LIN {X 0,Y 319.792,Z 522.033,A -85,B 0,C 180,E1 -15954.335,E2 -15954.335} C_VEL
LIN {X 0,Y 322.033,Z 507.948,A -85,B 0,C 180,E1 -15955.273,E2 -15955.273} C_VEL
LIN {X 0,Y 323.878,Z 494.069,A -85,B 0,C 180,E1 -15955.937,E2 -15955.937} C_VEL
LIN {X 0,Y 327.303,Z 451.829,A -85,B 0,C 180,E1 -15957.515,E2 -15957.515} C_VEL
LIN {X 0,Y 327.13,Z 436.75,A -85,B 0,C 180,E1 -15958.347,E2 -15958.347} C_VEL
LIN {X 0,Y 326.42,Z 425.043,A -85,B 0,C 180,E1 -15959.132,E2 -15959.132} C_VEL
LIN {X 0,Y 324.764,Z 409.047,A -85,B 0,C 180,E1 -15960.415,E2 -15960.415} C_VEL
LIN {X 0,Y 322.67,Z 394.757,A -85,B 0,C 180,E1 -15961.813,E2 -15961.813} C_VEL
LIN {X 0,Y 321.461,Z 387.953,A -85,B 0,C 180,E1 -15962.586,E2 -15962.586} C_VEL
LIN {X 0,Y 318.501,Z 381.059,A -85,B 0,C 180,E1 -15963.912,E2 -15963.912} C_VEL
LIN {X 0,Y 314.98,Z 373.335,A -85,B 0,C 180,E1 -15965.732,E2 -15965.732} C_VEL
LIN {X 0,Y 313.18,Z 366.557,A -85,B 0,C 180,E1 -15968.928,E2 -15968.928} C_VEL
LIN {X 0,Y 311.644,Z 361.486,A -85,B 0,C 180,E1 -15971.909,E2 -15971.909} C_VEL
LIN {X 0,Y 310.482,Z 357.991,A -85,B 0,C 180,E1 -15974.564,E2 -15974.564} C_VEL
LIN {X 0,Y 309.635,Z 355.475,A -85,B 0,C 180,E1 -15977.083,E2 -15977.083} C_VEL
LIN {X 0,Y 308.797,Z 353.363,A -85,B 0,C 180,E1 -15980.412,E2 -15980.412} C_VEL
LIN {X 0,Y 308.673,Z 352.451,A -85,B 0,C 180,E1 -15983.479,E2 -15983.479} C_VEL
LIN {X 0,Y 311.559,Z 355.007,A -85,B 0,C 180,E1 -15985.595,E2 -15985.595} C_VEL
LIN {X 0,Y 312.784,Z 355.997,A -85,B 0,C 180,E1 -15986.322,E2 -15986.322} C_VEL
LIN {X 0,Y 315.573,Z 358.678,A -85,B 0,C 180,E1 -15987.81,E2 -15987.81} C_VEL
LIN {X 0,Y 319.573,Z 362.862,A -85,B 0,C 180,E1 -15989.614,E2 -15989.614} C_VEL
LIN {X 0,Y 321.252,Z 365.21,A -85,B 0,C 180,E1 -15990.325,E2 -15990.325} C_VEL
LIN {X 0,Y 324.066,Z 369.646,A -85,B 0,C 180,E1 -15991.46,E2 -15991.46} C_VEL
LIN {X 0,Y 328.333,Z 376.83,A -85,B 0,C 180,E1 -15993.003,E2 -15993.003} C_VEL
LIN {X 0,Y 331.948,Z 384.05,A -85,B 0,C 180,E1 -15994.229,E2 -15994.229} C_VEL
LIN {X 0,Y 327.639,Z 429.139,A -85,B 0,C 180,E1 -15995.948,E2 -15995.948} C_VEL
LIN {X 0,Y 326.474,Z 447.037,A -85,B 0,C 180,E1 -15996.783,E2 -15996.783} C_VEL
LIN {X 0,Y 325.272,Z 459.562,A -85,B 0,C 180,E1 -15997.615,E2 -15997.615} C_VEL
LIN {X 0,Y 323.677,Z 471.852,A -85,B 0,C 180,E1 -15998.672,E2 -15998.672} C_VEL
LIN {X 0,Y 321.748,Z 483.617,A -85,B 0,C 180,E1 -15999.978,E2 -15999.978} C_VEL
LIN {X 0,Y 319.717,Z 494.029,A -85,B 0,C 180,E1 -16001.413,E2 -16001.413} C_VEL
LIN {X 0,Y 317.643,Z 503.088,A -85,B 0,C 180,E1 -16002.965,E2 -16002.965} C_VEL
LIN {X 0,Y 315.413,Z 511.843,A -85,B 0,C 180,E1 -16004.822,E2 -16004.822} C_VEL
LIN {X 0,Y 313.364,Z 518.904,A -85,B 0,C 180,E1 -16006.709,E2 -16006.709} C_VEL
LIN {X 0,Y 311.245,Z 525.34,A -85,B 0,C 180,E1 -16008.934,E2 -16008.934} C_VEL
LIN {X 0,Y 309.727,Z 529.542,A -85,B 0,C 180,E1 -16010.86,E2 -16010.86} C_VEL
LIN {X 0,Y 308.801,Z 531.727,A -85,B 0,C 180,E1 -16012.151,E2 -16012.151} C_VEL
LIN {X 0,Y 308.055,Z 533.416,A -85,B 0,C 180,E1 -16013.449,E2 -16013.449} C_VEL
LIN {X 0,Y 307.337,Z 534.702,A -85,B 0,C 180,E1 -16014.751,E2 -16014.751} C_VEL
LIN {X 0,Y 306.774,Z 535.536,A -85,B 0,C 180,E1 -16016.058,E2 -16016.058} C_VEL
LIN {X 0,Y 306.324,Z 535.911,A -85,B 0,C 180,E1 -16017.369,E2 -16017.369} C_VEL
LIN {X 0,Y 305.89,Z 535.895,A -85,B 0,C 180,E1 -16018.683,E2 -16018.683} C_VEL
LIN {X 0,Y 305.719,Z 535.443,A -85,B 0,C 180,E1 -16019.999,E2 -16019.999} C_VEL
LIN {X 0,Y 305.281,Z 534.566,A -85,B 0,C 180,E1 -16021.319,E2 -16021.319} C_VEL
LIN {X 0,Y 304.947,Z 533.258,A -85,B 0,C 180,E1 -16022.641,E2 -16022.641} C_VEL
LIN {X 0,Y 305.096,Z 530.427,A -85,B 0,C 180,E1 -16024.624,E2 -16024.624} C_VEL
LIN {X 0,Y 305.23,Z 526.556,A -85,B 0,C 180,E1 -16026.61,E2 -16026.61} C_VEL
LIN {X 0,Y 305.436,Z 520.675,A -85,B 0,C 180,E1 -16028.901,E2 -16028.901} C_VEL
LIN {X 0,Y 305.844,Z 513.952,A -85,B 0,C 180,E1 -16030.927,E2 -16030.927} C_VEL
LIN {X 0,Y 306.334,Z 505.75,A -85,B 0,C 180,E1 -16032.925,E2 -16032.925} C_VEL
LIN {X 0,Y 307.006,Z 497.416,A -85,B 0,C 180,E1 -16034.584,E2 -16034.584} C_VEL
LIN {X 0,Y 307.658,Z 486.376,A -85,B 0,C 180,E1 -16036.376,E2 -16036.376} C_VEL
LIN {X 0,Y 308.382,Z 476.01,A -85,B 0,C 180,E1 -16037.746,E2 -16037.746} C_VEL
LIN {X 0,Y 309.142,Z 463.45,A -85,B 0,C 180,E1 -16039.074,E2 -16039.074} C_VEL
LIN {X 0,Y 309.82,Z 450.341,A -85,B 0,C 180,E1 -16040.152,E2 -16040.152} C_VEL
LIN {X 0,Y 310.318,Z 435.654,A -85,B 0,C 180,E1 -16041.027,E2 -16041.027} C_VEL
LIN {X 0,Y 310.53,Z 421.083,A -85,B 0,C 180,E1 -16041.604,E2 -16041.604} C_VEL
LIN {X 0,Y 312.068,Z 364.546,A -85,B 0,C 180,E1 -16043.438,E2 -16043.438} C_VEL
LIN {X 0,Y 305.564,Z 343.422,A -85,B 0,C 180,E1 -16044.456,E2 -16044.456} C_VEL
LIN {X 0,Y 305.534,Z 343.424,A -85,B 0,C 180,E1 -16047.389,E2 -16047.389} C_VEL
LIN {X 0,Y 305.463,Z 343.433,A -85,B 0,C 180,E1 -16050.408,E2 -16050.408} C_VEL
LIN {X 0,Y 305.463,Z 343.432,A -85,B 0,C 180,E1 -16054.078,E2 -16054.078} C_VEL
LIN {X 0,Y 305.471,Z 343.436,A -85,B 0,C 180,E1 -16056.739,E2 -16056.739} C_VEL
LIN {X 0,Y 305.453,Z 343.437,A -85,B 0,C 180,E1 -16060.599,E2 -16060.599} C_VEL
LIN {X 0,Y 305.417,Z 343.441,A -85,B 0,C 180,E1 -16064.492,E2 -16064.492} C_VEL
LIN {X 0,Y 305.44,Z 343.436,A -85,B 0,C 180,E1 -16068.143,E2 -16068.143} C_VEL
LIN {X 0,Y 305.493,Z 343.428,A -85,B 0,C 180,E1 -16071.6,E2 -16071.6} C_VEL
LIN {X 0,Y 305.46,Z 343.435,A -85,B 0,C 180,E1 -16074.887,E2 -16074.887} C_VEL
LIN {X 0,Y 305.447,Z 343.437,A -85,B 0,C 180,E1 -16078.355,E2 -16078.355} C_VEL
LIN {X 0,Y 305.51,Z 343.428,A -85,B 0,C 180,E1 -16081.113,E2 -16081.113} C_VEL
LIN {X 0,Y 305.562,Z 343.421,A -85,B 0,C 180,E1 -16084.087,E2 -16084.087} C_VEL
LIN {X 0,Y 305.498,Z 343.432,A -85,B 0,C 180,E1 -16088.403,E2 -16088.403} C_VEL
LIN {X 0,Y 305.587,Z 343.417,A -85,B 0,C 180,E1 -16091.218,E2 -16091.218} C_VEL
LIN {X 0,Y 305.646,Z 343.409,A -85,B 0,C 180,E1 -16095.349,E2 -16095.349} C_VEL
LIN {X 0,Y 305.636,Z 343.41,A -85,B 0,C 180,E1 -16099.4,E2 -16099.4} C_VEL
LIN {X 0,Y 305.81,Z 343.391,A -85,B 0,C 180,E1 -16102.074,E2 -16102.074} C_VEL
LIN {X 0,Y 305.687,Z 343.407,A -85,B 0,C 180,E1 -16104.724,E2 -16104.724} C_VEL
LIN {X 0,Y 305.955,Z 343.373,A -85,B 0,C 180,E1 -16108.684,E2 -16108.684} C_VEL
LIN {X 0,Y 305.955,Z 343.371,A -85,B 0,C 180,E1 -16111.316,E2 -16111.316} C_VEL
LIN {X 0,Y 305.85,Z 343.387,A -85,B 0,C 180,E1 -16116.598,E2 -16116.598} C_VEL
LIN {X 0,Y 305.733,Z 343.398,A -85,B 0,C 180,E1 -16119.26,E2 -16119.26} C_VEL
LIN {X 0,Y 305.586,Z 343.417,A -85,B 0,C 180,E1 -16123.296,E2 -16123.296} C_VEL
LIN {X 0,Y 305.591,Z 343.419,A -85,B 0,C 180,E1 -16126.021,E2 -16126.021} C_VEL
LIN {X 0,Y 305.575,Z 343.418,A -85,B 0,C 180,E1 -16129.446,E2 -16129.446} C_VEL
LIN {X 0,Y 305.488,Z 343.429,A -85,B 0,C 180,E1 -16133.042,E2 -16133.042} C_VEL
LIN {X 0,Y 305.545,Z 343.427,A -85,B 0,C 180,E1 -16136.227,E2 -16136.227} C_VEL
LIN {X 0,Y 305.486,Z 343.429,A -85,B 0,C 180,E1 -16139.048,E2 -16139.048} C_VEL
LIN {X 0,Y 305.441,Z 343.439,A -85,B 0,C 180,E1 -16141.953,E2 -16141.953} C_VEL
LIN {X 0,Y 305.461,Z 343.432,A -85,B 0,C 180,E1 -16145.114,E2 -16145.114} C_VEL
LIN {X 0,Y 305.466,Z 343.434,A -85,B 0,C 180,E1 -16148.534,E2 -16148.534} C_VEL
LIN {X 0,Y 305.454,Z 343.434,A -85,B 0,C 180,E1 -16152.587,E2 -16152.587} C_VEL
LIN {X 0,Y 305.425,Z 343.44,A -85,B 0,C 180,E1 -16156.346,E2 -16156.346} C_VEL
LIN {X 0,Y 305.458,Z 343.437,A -85,B 0,C 180,E1 -16159.893,E2 -16159.893} C_VEL
LIN {X 0,Y 305.484,Z 343.432,A -85,B 0,C 180,E1 -16163.632,E2 -16163.632} C_VEL
LIN {X 0,Y 305.466,Z 343.433,A -85,B 0,C 180,E1 -16166.484,E2 -16166.484} C_VEL
LIN {X 0,Y 305.541,Z 343.424,A -85,B 0,C 180,E1 -16169.339,E2 -16169.339} C_VEL
LIN {X 0,Y 312.554,Z 364.965,A -85,B 0,C 180,E1 -16170.391,E2 -16170.391} C_VEL
LIN {X 0,Y 310.802,Z 429.878,A -85,B 0,C 180,E1 -16172.43,E2 -16172.43} C_VEL
LIN {X 0,Y 310.52,Z 443.041,A -85,B 0,C 180,E1 -16173.086,E2 -16173.086} C_VEL
LIN {X 0,Y 310.034,Z 453.965,A -85,B 0,C 180,E1 -16173.829,E2 -16173.829} C_VEL
LIN {X 0,Y 309.055,Z 459.424,A -85,B 0,C 180,E1 -16174.25,E2 -16174.25} C_VEL
LIN {X 0,Y 305.775,Z 467.979,A -85,B 0,C 180,E1 -16174.962,E2 -16174.962} C_VEL
LIN {X 0,Y 302.456,Z 476.194,A -85,B 0,C 180,E1 -16175.79,E2 -16175.79} C_VEL
LIN {X 0,Y 301.421,Z 481.034,A -85,B 0,C 180,E1 -16176.383,E2 -16176.383} C_VEL
LIN {X 0,Y 300.653,Z 491.112,A -85,B 0,C 180,E1 -16177.857,E2 -16177.857} C_VEL
LIN {X 0,Y 299.856,Z 501.018,A -85,B 0,C 180,E1 -16179.64,E2 -16179.64} C_VEL
LIN {X 0,Y 299.223,Z 509.544,A -85,B 0,C 180,E1 -16181.514,E2 -16181.514} C_VEL
LIN {X 0,Y 298.636,Z 517.147,A -85,B 0,C 180,E1 -16183.597,E2 -16183.597} C_VEL
LIN {X 0,Y 298.286,Z 523.209,A -85,B 0,C 180,E1 -16185.677,E2 -16185.677} C_VEL
LIN {X 0,Y 298.048,Z 527.957,A -85,B 0,C 180,E1 -16187.748,E2 -16187.748} C_VEL
LIN {X 0,Y 298.032,Z 530.453,A -85,B 0,C 180,E1 -16189.127,E2 -16189.127} C_VEL
LIN {X 0,Y 298.226,Z 533.945,A -85,B 0,C 180,E1 -16191.803,E2 -16191.803} C_VEL
LIN {X 0,Y 298.414,Z 535.09,A -85,B 0,C 180,E1 -16193.238,E2 -16193.238} C_VEL
LIN {X 0,Y 298.541,Z 535.761,A -85,B 0,C 180,E1 -16194.597,E2 -16194.597} C_VEL
LIN {X 0,Y 298.905,Z 536.001,A -85,B 0,C 180,E1 -16195.956,E2 -16195.956} C_VEL
LIN {X 0,Y 299.354,Z 535.769,A -85,B 0,C 180,E1 -16197.309,E2 -16197.309} C_VEL
LIN {X 0,Y 299.866,Z 535.126,A -85,B 0,C 180,E1 -16198.658,E2 -16198.658} C_VEL
LIN {X 0,Y 300.486,Z 534.078,A -85,B 0,C 180,E1 -16200.001,E2 -16200.001} C_VEL
LIN {X 0,Y 301.229,Z 532.545,A -85,B 0,C 180,E1 -16201.338,E2 -16201.338} C_VEL
LIN {X 0,Y 302.893,Z 528.394,A -85,B 0,C 180,E1 -16203.857,E2 -16203.857} C_VEL
LIN {X 0,Y 304.578,Z 523.469,A -85,B 0,C 180,E1 -16205.961,E2 -16205.961} C_VEL
LIN {X 0,Y 306.754,Z 516.45,A -85,B 0,C 180,E1 -16208.233,E2 -16208.233} C_VEL
LIN {X 0,Y 308.88,Z 508.771,A -85,B 0,C 180,E1 -16210.157,E2 -16210.157} C_VEL
LIN {X 0,Y 310.744,Z 500.928,A -85,B 0,C 180,E1 -16211.745,E2 -16211.745} C_VEL
LIN {X 0,Y 313.057,Z 490.377,A -85,B 0,C 180,E1 -16213.469,E2 -16213.469} C_VEL
LIN {X 0,Y 315.044,Z 479.613,A -85,B 0,C 180,E1 -16214.866,E2 -16214.866} C_VEL
LIN {X 0,Y 316.877,Z 467.593,A -85,B 0,C 180,E1 -16216.096,E2 -16216.096} C_VEL
LIN {X 0,Y 318.282,Z 454.819,A -85,B 0,C 180,E1 -16217.109,E2 -16217.109} C_VEL
LIN {X 0,Y 319.298,Z 441.159,A -85,B 0,C 180,E1 -16217.912,E2 -16217.912} C_VEL
LIN {X 0,Y 320.981,Z 415.483,A -85,B 0,C 180,E1 -16218.921,E2 -16218.921} C_VEL
LIN {X 0,Y 323.739,Z 383.791,A -85,B 0,C 180,E1 -16220.056,E2 -16220.056} C_VEL
LIN {X 0,Y 318.843,Z 374.597,A -85,B 0,C 180,E1 -16221.566,E2 -16221.566} C_VEL
LIN {X 0,Y 314.171,Z 366.92,A -85,B 0,C 180,E1 -16223.133,E2 -16223.133} C_VEL
LIN {X 0,Y 311.791,Z 363.309,A -85,B 0,C 180,E1 -16223.977,E2 -16223.977} C_VEL
LIN {X 0,Y 309.279,Z 359.484,A -85,B 0,C 180,E1 -16224.966,E2 -16224.966} C_VEL
LIN {X 0,Y 307.001,Z 356.45,A -85,B 0,C 180,E1 -16225.897,E2 -16225.897} C_VEL
LIN {X 0,Y 306.138,Z 354.997,A -85,B 0,C 180,E1 -16226.305,E2 -16226.305} C_VEL
LIN {X 0,Y 303.664,Z 352.303,A -85,B 0,C 180,E1 -16227.398,E2 -16227.398} C_VEL
LIN {X 0,Y 302.59,Z 349.926,A -85,B 0,C 180,E1 -16228.042,E2 -16228.042} C_VEL
LIN {X 0,Y 299.804,Z 347.798,A -85,B 0,C 180,E1 -16229.443,E2 -16229.443} C_VEL
LIN {X 0,Y 298.576,Z 345.283,A -85,B 0,C 180,E1 -16230.322,E2 -16230.322} C_VEL
LIN {X 0,Y 298.376,Z 344.317,A -85,B 0,C 180,E1 -16230.572,E2 -16230.572} C_VEL
LIN {X 0,Y 298.432,Z 344.308,A -85,B 0,C 180,E1 -16234.488,E2 -16234.488} C_VEL
LIN {X 0,Y 298.392,Z 344.31,A -85,B 0,C 180,E1 -16237.762,E2 -16237.762} C_VEL
LIN {X 0,Y 298.351,Z 344.315,A -85,B 0,C 180,E1 -16241.268,E2 -16241.268} C_VEL
LIN {X 0,Y 298.358,Z 344.32,A -85,B 0,C 180,E1 -16245.035,E2 -16245.035} C_VEL
LIN {X 0,Y 298.385,Z 344.332,A -85,B 0,C 180,E1 -16246.621,E2 -16246.621} C_VEL
LIN {X 0,Y 299.056,Z 346.56,A -85,B 0,C 180,E1 -16247.754,E2 -16247.754} C_VEL
LIN {X 0,Y 301.947,Z 350.438,A -85,B 0,C 180,E1 -16250.184,E2 -16250.184} C_VEL
LIN {X 0,Y 305.332,Z 355.742,A -85,B 0,C 180,E1 -16252.504,E2 -16252.504} C_VEL
LIN {X 0,Y 307.435,Z 358.849,A -85,B 0,C 180,E1 -16253.69,E2 -16253.69} C_VEL
LIN {X 0,Y 309.769,Z 368.647,A -85,B 0,C 180,E1 -16255.644,E2 -16255.644} C_VEL
LIN {X 0,Y 312.563,Z 376.409,A -85,B 0,C 180,E1 -16256.91,E2 -16256.91} C_VEL
LIN {X 0,Y 314.336,Z 382.808,A -85,B 0,C 180,E1 -16257.746,E2 -16257.746} C_VEL
LIN {X 0,Y 316.181,Z 399.413,A -85,B 0,C 180,E1 -16259.138,E2 -16259.138} C_VEL
LIN {X 0,Y 317.764,Z 420.425,A -85,B 0,C 180,E1 -16260.619,E2 -16260.619} C_VEL
LIN {X 0,Y 318.753,Z 439.399,A -85,B 0,C 180,E1 -16261.791,E2 -16261.791} C_VEL
LIN {X 0,Y 318.965,Z 455.73,A -85,B 0,C 180,E1 -16262.623,E2 -16262.623} C_VEL
LIN {X 0,Y 315.657,Z 497.328,A -85,B 0,C 180,E1 -16264.135,E2 -16264.135} C_VEL
LIN {X 0,Y 313.836,Z 511.992,A -85,B 0,C 180,E1 -16264.907,E2 -16264.907} C_VEL
LIN {X 0,Y 311.504,Z 525.439,A -85,B 0,C 180,E1 -16265.862,E2 -16265.862} C_VEL
LIN {X 0,Y 308.965,Z 538.23,A -85,B 0,C 180,E1 -16267.074,E2 -16267.074} C_VEL
LIN {X 0,Y 306.449,Z 549.812,A -85,B 0,C 180,E1 -16268.473,E2 -16268.473} C_VEL
LIN {X 0,Y 304.162,Z 560.405,A -85,B 0,C 180,E1 -16270.073,E2 -16270.073} C_VEL
LIN {X 0,Y 302.001,Z 569.208,A -85,B 0,C 180,E1 -16271.689,E2 -16271.689} C_VEL
LIN {X 0,Y 300.09,Z 577.969,A -85,B 0,C 180,E1 -16273.678,E2 -16273.678} C_VEL
LIN {X 0,Y 298.705,Z 585.204,A -85,B 0,C 180,E1 -16275.697,E2 -16275.697} C_VEL
LIN {X 0,Y 297.796,Z 591.06,A -85,B 0,C 180,E1 -16277.737,E2 -16277.737} C_VEL
LIN {X 0,Y 297.24,Z 595.727,A -85,B 0,C 180,E1 -16279.785,E2 -16279.785} C_VEL
LIN {X 0,Y 297.071,Z 599.337,A -85,B 0,C 180,E1 -16281.839,E2 -16281.839} C_VEL
LIN {X 0,Y 297.21,Z 601.262,A -85,B 0,C 180,E1 -16283.297,E2 -16283.297} C_VEL
LIN {X 0,Y 297.556,Z 603.522,A -85,B 0,C 180,E1 -16285.937,E2 -16285.937} C_VEL
LIN {X 0,Y 297.744,Z 603.993,A -85,B 0,C 180,E1 -16287.294,E2 -16287.294} C_VEL
LIN {X 0,Y 297.946,Z 604.017,A -85,B 0,C 180,E1 -16288.648,E2 -16288.648} C_VEL
LIN {X 0,Y 298.065,Z 604.583,A -85,B 0,C 180,E1 -16290,E2 -16290} C_VEL
LIN {X 0,Y 297.82,Z 605.131,A -85,B 0,C 180,E1 -16291.352,E2 -16291.352} C_VEL
LIN {X 0,Y 297.655,Z 605.194,A -85,B 0,C 180,E1 -16292.706,E2 -16292.706} C_VEL
LIN {X 0,Y 297.475,Z 604.807,A -85,B 0,C 180,E1 -16294.064,E2 -16294.064} C_VEL
LIN {X 0,Y 297.135,Z 602.937,A -85,B 0,C 180,E1 -16296.578,E2 -16296.578} C_VEL
LIN {X 0,Y 297.035,Z 599.978,A -85,B 0,C 180,E1 -16298.847,E2 -16298.847} C_VEL
LIN {X 0,Y 297.276,Z 596.23,A -85,B 0,C 180,E1 -16300.902,E2 -16300.902} C_VEL
LIN {X 0,Y 298.054,Z 591.434,A -85,B 0,C 180,E1 -16302.944,E2 -16302.944} C_VEL
LIN {X 0,Y 299.235,Z 585.477,A -85,B 0,C 180,E1 -16304.972,E2 -16304.972} C_VEL
LIN {X 0,Y 300.786,Z 578.223,A -85,B 0,C 180,E1 -16306.982,E2 -16306.982} C_VEL
LIN {X 0,Y 302.901,Z 569.407,A -85,B 0,C 180,E1 -16308.955,E2 -16308.955} C_VEL
LIN {X 0,Y 305.618,Z 558.724,A -85,B 0,C 180,E1 -16310.882,E2 -16310.882} C_VEL
LIN {X 0,Y 308.258,Z 547.881,A -85,B 0,C 180,E1 -16312.45,E2 -16312.45} C_VEL
LIN {X 0,Y 311.026,Z 536.102,A -85,B 0,C 180,E1 -16313.823,E2 -16313.823} C_VEL
LIN {X 0,Y 313.81,Z 523.137,A -85,B 0,C 180,E1 -16315.006,E2 -16315.006} C_VEL
LIN {X 0,Y 316.353,Z 508.822,A -85,B 0,C 180,E1 -16316.025,E2 -16316.025} C_VEL
LIN {X 0,Y 318.487,Z 494.166,A -85,B 0,C 180,E1 -16316.763,E2 -16316.763} C_VEL
LIN {X 0,Y 322.192,Z 452.495,A -85,B 0,C 180,E1 -16318.383,E2 -16318.383} C_VEL
LIN {X 0,Y 322.153,Z 438.563,A -85,B 0,C 180,E1 -16319.181,E2 -16319.181} C_VEL
LIN {X 0,Y 321.531,Z 426.086,A -85,B 0,C 180,E1 -16320.054,E2 -16320.054} C_VEL
LIN {X 0,Y 320.216,Z 411.813,A -85,B 0,C 180,E1 -16321.256,E2 -16321.256} C_VEL
LIN {X 0,Y 318.449,Z 398.178,A -85,B 0,C 180,E1 -16322.636,E2 -16322.636} C_VEL
LIN {X 0,Y 317.494,Z 392.313,A -85,B 0,C 180,E1 -16323.332,E2 -16323.332} C_VEL
LIN {X 0,Y 315.207,Z 386.547,A -85,B 0,C 180,E1 -16324.471,E2 -16324.471} C_VEL
LIN {X 0,Y 311.613,Z 378.51,A -85,B 0,C 180,E1 -16326.441,E2 -16326.441} C_VEL
LIN {X 0,Y 306.703,Z 368.661,A -85,B 0,C 180,E1 -16329.912,E2 -16329.912} C_VEL
LIN {X 0,Y 306.143,Z 367.078,A -85,B 0,C 180,E1 -16330.749,E2 -16330.749} C_VEL
LIN {X 0,Y 304.853,Z 362.75,A -85,B 0,C 180,E1 -16333.758,E2 -16333.758} C_VEL
LIN {X 0,Y 303.957,Z 360.236,A -85,B 0,C 180,E1 -16336.079,E2 -16336.079} C_VEL
LIN {X 0,Y 303.279,Z 358.239,A -85,B 0,C 180,E1 -16338.653,E2 -16338.653} C_VEL
LIN {X 0,Y 304.892,Z 358.916,A -85,B 0,C 180,E1 -16341.603,E2 -16341.603} C_VEL
LIN {X 0,Y 306.92,Z 359.438,A -85,B 0,C 180,E1 -16343.461,E2 -16343.461} C_VEL
LIN {X 0,Y 309.723,Z 361.859,A -85,B 0,C 180,E1 -16345.546,E2 -16345.546} C_VEL
LIN {X 0,Y 310.688,Z 362.763,A -85,B 0,C 180,E1 -16346.149,E2 -16346.149} C_VEL
LIN {X 0,Y 313.943,Z 366.078,A -85,B 0,C 180,E1 -16347.929,E2 -16347.929} C_VEL
LIN {X 0,Y 317.111,Z 369.474,A -85,B 0,C 180,E1 -16349.385,E2 -16349.385} C_VEL
LIN {X 0,Y 320.546,Z 374.9,A -85,B 0,C 180,E1 -16350.889,E2 -16350.889} C_VEL
LIN {X 0,Y 325.155,Z 383.081,A -85,B 0,C 180,E1 -16352.675,E2 -16352.675} C_VEL
LIN {X 0,Y 327.04,Z 386.949,A -85,B 0,C 180,E1 -16353.365,E2 -16353.365} C_VEL
LIN {X 0,Y 322.581,Z 431.149,A -85,B 0,C 180,E1 -16355.117,E2 -16355.117} C_VEL
LIN {X 0,Y 321.307,Z 448.525,A -85,B 0,C 180,E1 -16355.959,E2 -16355.959} C_VEL
LIN {X 0,Y 319.906,Z 461.798,A -85,B 0,C 180,E1 -16356.877,E2 -16356.877} C_VEL
LIN {X 0,Y 318.194,Z 473.732,A -85,B 0,C 180,E1 -16357.945,E2 -16357.945} C_VEL
LIN {X 0,Y 315.87,Z 486.528,A -85,B 0,C 180,E1 -16359.421,E2 -16359.421} C_VEL
LIN {X 0,Y 313.589,Z 496.975,A -85,B 0,C 180,E1 -16360.952,E2 -16360.952} C_VEL
LIN {X 0,Y 311.301,Z 506.046,A -85,B 0,C 180,E1 -16362.594,E2 -16362.594} C_VEL
LIN {X 0,Y 308.948,Z 514.418,A -85,B 0,C 180,E1 -16364.496,E2 -16364.496} C_VEL
LIN {X 0,Y 306.784,Z 521.167,A -85,B 0,C 180,E1 -16366.419,E2 -16366.419} C_VEL
LIN {X 0,Y 304.553,Z 527.32,A -85,B 0,C 180,E1 -16368.687,E2 -16368.687} C_VEL
LIN {X 0,Y 302.931,Z 531.282,A -85,B 0,C 180,E1 -16370.653,E2 -16370.653} C_VEL
LIN {X 0,Y 301.943,Z 533.311,A -85,B 0,C 180,E1 -16371.971,E2 -16371.971} C_VEL
LIN {X 0,Y 301.156,Z 534.899,A -85,B 0,C 180,E1 -16373.299,E2 -16373.299} C_VEL
LIN {X 0,Y 300.422,Z 536.041,A -85,B 0,C 180,E1 -16374.63,E2 -16374.63} C_VEL
LIN {X 0,Y 299.801,Z 536.727,A -85,B 0,C 180,E1 -16375.967,E2 -16375.967} C_VEL
LIN {X 0,Y 299.322,Z 537.007,A -85,B 0,C 180,E1 -16377.308,E2 -16377.308} C_VEL
LIN {X 0,Y 298.868,Z 536.884,A -85,B 0,C 180,E1 -16378.652,E2 -16378.652} C_VEL
LIN {X 0,Y 298.661,Z 536.273,A -85,B 0,C 180,E1 -16379.999,E2 -16379.999} C_VEL
LIN {X 0,Y 298.206,Z 535.285,A -85,B 0,C 180,E1 -16381.35,E2 -16381.35} C_VEL
LIN {X 0,Y 297.897,Z 533.876,A -85,B 0,C 180,E1 -16382.704,E2 -16382.704} C_VEL
LIN {X 0,Y 298.045,Z 530.856,A -85,B 0,C 180,E1 -16384.733,E2 -16384.733} C_VEL
LIN {X 0,Y 298.17,Z 526.787,A -85,B 0,C 180,E1 -16386.768,E2 -16386.768} C_VEL
LIN {X 0,Y 298.395,Z 520.595,A -85,B 0,C 180,E1 -16389.113,E2 -16389.113} C_VEL
LIN {X 0,Y 298.821,Z 513.638,A -85,B 0,C 180,E1 -16391.188,E2 -16391.188} C_VEL
LIN {X 0,Y 299.347,Z 505.108,A -85,B 0,C 180,E1 -16393.232,E2 -16393.232} C_VEL
LIN {X 0,Y 300.02,Z 496.423,A -85,B 0,C 180,E1 -16394.932,E2 -16394.932} C_VEL
LIN {X 0,Y 300.66,Z 486.195,A -85,B 0,C 180,E1 -16396.587,E2 -16396.587} C_VEL
LIN {X 0,Y 301.393,Z 475.47,A -85,B 0,C 180,E1 -16397.996,E2 -16397.996} C_VEL
LIN {X 0,Y 302.192,Z 462.57,A -85,B 0,C 180,E1 -16399.354,E2 -16399.354} C_VEL
LIN {X 0,Y 302.828,Z 450.061,A -85,B 0,C 180,E1 -16400.372,E2 -16400.372} C_VEL
LIN {X 0,Y 303.322,Z 435.92,A -85,B 0,C 180,E1 -16401.224,E2 -16401.224} C_VEL
LIN {X 0,Y 303.519,Z 419.912,A -85,B 0,C 180,E1 -16401.859,E2 -16401.859} C_VEL
LIN {X 0,Y 305.102,Z 365.716,A -85,B 0,C 180,E1 -16403.677,E2 -16403.677} C_VEL
LIN {X 0,Y 298.524,Z 344.301,A -85,B 0,C 180,E1 -16404.726,E2 -16404.726} C_VEL
LIN {X 0,Y 298.469,Z 344.303,A -85,B 0,C 180,E1 -16408.094,E2 -16408.094} C_VEL
LIN {X 0,Y 298.394,Z 344.318,A -85,B 0,C 180,E1 -16412.799,E2 -16412.799} C_VEL
LIN {X 0,Y 298.443,Z 344.312,A -85,B 0,C 180,E1 -16416.806,E2 -16416.806} C_VEL
LIN {X 0,Y 298.386,Z 344.316,A -85,B 0,C 180,E1 -16421.087,E2 -16421.087} C_VEL
LIN {X 0,Y 298.386,Z 344.316,A -85,B 0,C 180,E1 -16425.041,E2 -16425.041} C_VEL
LIN {X 0,Y 298.386,Z 344.317,A -85,B 0,C 180,E1 -16428.912,E2 -16428.912} C_VEL
LIN {X 0,Y 298.462,Z 344.305,A -85,B 0,C 180,E1 -16433.187,E2 -16433.187} C_VEL
LIN {X 0,Y 298.392,Z 344.314,A -85,B 0,C 180,E1 -16437.199,E2 -16437.199} C_VEL
LIN {X 0,Y 298.424,Z 344.314,A -85,B 0,C 180,E1 -16440.616,E2 -16440.616} C_VEL
LIN {X 0,Y 298.474,Z 344.302,A -85,B 0,C 180,E1 -16443.477,E2 -16443.477} C_VEL
LIN {X 0,Y 298.433,Z 344.312,A -85,B 0,C 180,E1 -16446.697,E2 -16446.697} C_VEL
LIN {X 0,Y 298.537,Z 344.298,A -85,B 0,C 180,E1 -16450.757,E2 -16450.757} C_VEL
LIN {X 0,Y 298.59,Z 344.29,A -85,B 0,C 180,E1 -16454.995,E2 -16454.995} C_VEL
LIN {X 0,Y 298.591,Z 344.289,A -85,B 0,C 180,E1 -16459.147,E2 -16459.147} C_VEL
LIN {X 0,Y 298.756,Z 344.268,A -85,B 0,C 180,E1 -16461.886,E2 -16461.886} C_VEL
LIN {X 0,Y 298.658,Z 344.284,A -85,B 0,C 180,E1 -16464.599,E2 -16464.599} C_VEL
LIN {X 0,Y 298.921,Z 344.25,A -85,B 0,C 180,E1 -16468.653,E2 -16468.653} C_VEL
LIN {X 0,Y 298.921,Z 344.247,A -85,B 0,C 180,E1 -16471.347,E2 -16471.347} C_VEL
LIN {X 0,Y 298.795,Z 344.264,A -85,B 0,C 180,E1 -16476.754,E2 -16476.754} C_VEL
LIN {X 0,Y 298.678,Z 344.277,A -85,B 0,C 180,E1 -16479.481,E2 -16479.481} C_VEL
LIN {X 0,Y 298.55,Z 344.294,A -85,B 0,C 180,E1 -16483.616,E2 -16483.616} C_VEL
LIN {X 0,Y 298.546,Z 344.297,A -85,B 0,C 180,E1 -16486.409,E2 -16486.409} C_VEL
LIN {X 0,Y 298.51,Z 344.299,A -85,B 0,C 180,E1 -16489.656,E2 -16489.656} C_VEL
LIN {X 0,Y 298.455,Z 344.306,A -85,B 0,C 180,E1 -16493.598,E2 -16493.598} C_VEL
LIN {X 0,Y 298.487,Z 344.303,A -85,B 0,C 180,E1 -16496.575,E2 -16496.575} C_VEL
LIN {X 0,Y 298.415,Z 344.311,A -85,B 0,C 180,E1 -16499.642,E2 -16499.642} C_VEL
LIN {X 0,Y 298.394,Z 344.313,A -85,B 0,C 180,E1 -16502.801,E2 -16502.801} C_VEL
LIN {X 0,Y 298.463,Z 344.305,A -85,B 0,C 180,E1 -16506.813,E2 -16506.813} C_VEL
LIN {X 0,Y 298.386,Z 344.313,A -85,B 0,C 180,E1 -16511.088,E2 -16511.088} C_VEL
LIN {X 0,Y 298.398,Z 344.312,A -85,B 0,C 180,E1 -16513.104,E2 -16513.104} C_VEL
LIN {X 0,Y 298.402,Z 344.312,A -85,B 0,C 180,E1 -16516.922,E2 -16516.922} C_VEL
LIN {X 0,Y 298.415,Z 344.309,A -85,B 0,C 180,E1 -16521.005,E2 -16521.005} C_VEL
LIN {X 0,Y 298.421,Z 344.314,A -85,B 0,C 180,E1 -16523.931,E2 -16523.931} C_VEL
LIN {X 0,Y 298.397,Z 344.317,A -85,B 0,C 180,E1 -16527.984,E2 -16527.984} C_VEL
LIN {X 0,Y 298.473,Z 344.304,A -85,B 0,C 180,E1 -16529.046,E2 -16529.046} C_VEL
LIN {X 0,Y 305.674,Z 367.027,A -85,B 0,C 180,E1 -16530.162,E2 -16530.162} C_VEL
LIN {X 0,Y 303.834,Z 430.008,A -85,B 0,C 180,E1 -16532.195,E2 -16532.195} C_VEL
LIN {X 0,Y 303.545,Z 443.656,A -85,B 0,C 180,E1 -16532.883,E2 -16532.883} C_VEL
LIN {X 0,Y 302.819,Z 458.173,A -85,B 0,C 180,E1 -16533.928,E2 -16533.928} C_VEL
LIN {X 0,Y 302.172,Z 470.383,A -85,B 0,C 180,E1 -16535.105,E2 -16535.105} C_VEL
LIN {X 0,Y 301.421,Z 481.034,A -85,B 0,C 180,E1 -16536.383,E2 -16536.383} C_VEL
LIN {X 0,Y 300.394,Z 485.82,A -85,B 0,C 180,E1 -16537.014,E2 -16537.014} C_VEL
LIN {X 0,Y 297.068,Z 493.295,A -85,B 0,C 180,E1 -16538.087,E2 -16538.087} C_VEL
LIN {X 0,Y 293.692,Z 500.271,A -85,B 0,C 180,E1 -16539.29,E2 -16539.29} C_VEL
LIN {X 0,Y 292.605,Z 504.276,A -85,B 0,C 180,E1 -16540.116,E2 -16540.116} C_VEL
LIN {X 0,Y 291.93,Z 512.662,A -85,B 0,C 180,E1 -16542.125,E2 -16542.125} C_VEL
LIN {X 0,Y 291.454,Z 519.889,A -85,B 0,C 180,E1 -16544.26,E2 -16544.26} C_VEL
LIN {X 0,Y 291.1,Z 526.386,A -85,B 0,C 180,E1 -16546.741,E2 -16546.741} C_VEL
LIN {X 0,Y 290.978,Z 530.616,A -85,B 0,C 180,E1 -16548.86,E2 -16548.86} C_VEL
LIN {X 0,Y 291.026,Z 532.803,A -85,B 0,C 180,E1 -16550.268,E2 -16550.268} C_VEL
LIN {X 0,Y 291.165,Z 534.575,A -85,B 0,C 180,E1 -16551.749,E2 -16551.749} C_VEL
LIN {X 0,Y 291.338,Z 535.763,A -85,B 0,C 180,E1 -16553.073,E2 -16553.073} C_VEL
LIN {X 0,Y 291.491,Z 536.584,A -85,B 0,C 180,E1 -16554.466,E2 -16554.466} C_VEL
LIN {X 0,Y 291.829,Z 536.954,A -85,B 0,C 180,E1 -16555.858,E2 -16555.858} C_VEL
LIN {X 0,Y 292.323,Z 536.91,A -85,B 0,C 180,E1 -16557.245,E2 -16557.245} C_VEL
LIN {X 0,Y 292.845,Z 536.434,A -85,B 0,C 180,E1 -16558.625,E2 -16558.625} C_VEL
LIN {X 0,Y 293.496,Z 535.499,A -85,B 0,C 180,E1 -16560.001,E2 -16560.001} C_VEL
LIN {X 0,Y 294.26,Z 534.151,A -85,B 0,C 180,E1 -16561.369,E2 -16561.369} C_VEL
LIN {X 0,Y 295.777,Z 530.885,A -85,B 0,C 180,E1 -16563.643,E2 -16563.643} C_VEL
LIN {X 0,Y 297.783,Z 525.74,A -85,B 0,C 180,E1 -16566.097,E2 -16566.097} C_VEL
LIN {X 0,Y 299.702,Z 520.171,A -85,B 0,C 180,E1 -16568.089,E2 -16568.089} C_VEL
LIN {X 0,Y 301.907,Z 513.11,A -85,B 0,C 180,E1 -16570.055,E2 -16570.055} C_VEL
LIN {X 0,Y 304.255,Z 504.47,A -85,B 0,C 180,E1 -16571.999,E2 -16571.999} C_VEL
LIN {X 0,Y 306.694,Z 494.511,A -85,B 0,C 180,E1 -16573.754,E2 -16573.754} C_VEL
LIN {X 0,Y 308.712,Z 484.518,A -85,B 0,C 180,E1 -16575.178,E2 -16575.178} C_VEL
LIN {X 0,Y 310.886,Z 472.003,A -85,B 0,C 180,E1 -16576.584,E2 -16576.584} C_VEL
LIN {X 0,Y 312.568,Z 459.587,A -85,B 0,C 180,E1 -16577.671,E2 -16577.671} C_VEL
LIN {X 0,Y 313.877,Z 445.237,A -85,B 0,C 180,E1 -16578.607,E2 -16578.607} C_VEL
LIN {X 0,Y 315.145,Z 425.429,A -85,B 0,C 180,E1 -16579.459,E2 -16579.459} C_VEL
LIN {X 0,Y 318.617,Z 386.676,A -85,B 0,C 180,E1 -16580.919,E2 -16580.919} C_VEL
LIN {X 0,Y 314.922,Z 379.654,A -85,B 0,C 180,E1 -16582.133,E2 -16582.133} C_VEL
LIN {X 0,Y 310.199,Z 371.685,A -85,B 0,C 180,E1 -16583.818,E2 -16583.818} C_VEL
LIN {X 0,Y 306.112,Z 365.369,A -85,B 0,C 180,E1 -16585.458,E2 -16585.458} C_VEL
LIN {X 0,Y 303.794,Z 361.887,A -85,B 0,C 180,E1 -16586.512,E2 -16586.512} C_VEL
LIN {X 0,Y 300.726,Z 357.957,A -85,B 0,C 180,E1 -16588.005,E2 -16588.005} C_VEL
LIN {X 0,Y 299.846,Z 356.294,A -85,B 0,C 180,E1 -16588.529,E2 -16588.529} C_VEL
LIN {X 0,Y 297.233,Z 353.82,A -85,B 0,C 180,E1 -16589.993,E2 -16589.993} C_VEL
LIN {X 0,Y 295.994,Z 350.978,A -85,B 0,C 180,E1 -16590.985,E2 -16590.985} C_VEL
LIN {X 0,Y 293.06,Z 349.016,A -85,B 0,C 180,E1 -16593.184,E2 -16593.184} C_VEL
LIN {X 0,Y 291.84,Z 346.98,A -85,B 0,C 180,E1 -16594.72,E2 -16594.72} C_VEL
LIN {X 0,Y 291.505,Z 345.918,A -85,B 0,C 180,E1 -16597.286,E2 -16597.286} C_VEL
LIN {X 0,Y 291.472,Z 346.073,A -85,B 0,C 180,E1 -16599.503,E2 -16599.503} C_VEL
LIN {X 0,Y 291.977,Z 347.485,A -85,B 0,C 180,E1 -16602.375,E2 -16602.375} C_VEL
LIN {X 0,Y 294.632,Z 350.347,A -85,B 0,C 180,E1 -16606.231,E2 -16606.231} C_VEL
LIN {X 0,Y 296.366,Z 353.961,A -85,B 0,C 180,E1 -16608.394,E2 -16608.394} C_VEL
LIN {X 0,Y 298.098,Z 356.087,A -85,B 0,C 180,E1 -16609.746,E2 -16609.746} C_VEL
LIN {X 0,Y 301.014,Z 360.643,A -85,B 0,C 180,E1 -16611.843,E2 -16611.843} C_VEL
LIN {X 0,Y 303.562,Z 365.1,A -85,B 0,C 180,E1 -16613.437,E2 -16613.437} C_VEL
LIN {X 0,Y 308.519,Z 380.45,A -85,B 0,C 180,E1 -16616.134,E2 -16616.134} C_VEL
LIN {X 0,Y 310.044,Z 386.463,A -85,B 0,C 180,E1 -16616.935,E2 -16616.935} C_VEL
LIN {X 0,Y 311.507,Z 402.284,A -85,B 0,C 180,E1 -16618.304,E2 -16618.304} C_VEL
LIN {X 0,Y 312.913,Z 423.75,A -85,B 0,C 180,E1 -16619.864,E2 -16619.864} C_VEL
LIN {X 0,Y 313.653,Z 442.028,A -85,B 0,C 180,E1 -16621.012,E2 -16621.012} C_VEL
LIN {X 0,Y 313.631,Z 457.032,A -85,B 0,C 180,E1 -16621.795,E2 -16621.795} C_VEL
LIN {X 0,Y 310.214,Z 496.855,A -85,B 0,C 180,E1 -16623.284,E2 -16623.284} C_VEL
LIN {X 0,Y 308.274,Z 511.102,A -85,B 0,C 180,E1 -16624.059,E2 -16624.059} C_VEL
LIN {X 0,Y 305.858,Z 524.313,A -85,B 0,C 180,E1 -16625.025,E2 -16625.025} C_VEL
LIN {X 0,Y 302.832,Z 538.458,A -85,B 0,C 180,E1 -16626.401,E2 -16626.401} C_VEL
LIN {X 0,Y 300.183,Z 549.805,A -85,B 0,C 180,E1 -16627.819,E2 -16627.819} C_VEL
LIN {X 0,Y 297.995,Z 559.161,A -85,B 0,C 180,E1 -16629.282,E2 -16629.282} C_VEL
LIN {X 0,Y 295.281,Z 569.55,A -85,B 0,C 180,E1 -16631.257,E2 -16631.257} C_VEL
LIN {X 0,Y 293.26,Z 578.056,A -85,B 0,C 180,E1 -16633.286,E2 -16633.286} C_VEL
LIN {X 0,Y 291.804,Z 585.009,A -85,B 0,C 180,E1 -16635.351,E2 -16635.351} C_VEL
LIN {X 0,Y 290.816,Z 590.69,A -85,B 0,C 180,E1 -16637.438,E2 -16637.438} C_VEL
LIN {X 0,Y 290.178,Z 595.212,A -85,B 0,C 180,E1 -16639.534,E2 -16639.534} C_VEL
LIN {X 0,Y 289.99,Z 598.677,A -85,B 0,C 180,E1 -16641.639,E2 -16641.639} C_VEL
LIN {X 0,Y 290.127,Z 600.741,A -85,B 0,C 180,E1 -16643.308,E2 -16643.308} C_VEL
LIN {X 0,Y 290.485,Z 602.623,A -85,B 0,C 180,E1 -16645.837,E2 -16645.837} C_VEL
LIN {X 0,Y 290.687,Z 603.029,A -85,B 0,C 180,E1 -16647.228,E2 -16647.228} C_VEL
LIN {X 0,Y 290.907,Z 603,A -85,B 0,C 180,E1 -16648.615,E2 -16648.615} C_VEL
LIN {X 0,Y 291.064,Z 603.388,A -85,B 0,C 180,E1 -16650,E2 -16650} C_VEL
LIN {X 0,Y 290.8,Z 604.013,A -85,B 0,C 180,E1 -16651.385,E2 -16651.385} C_VEL
LIN {X 0,Y 290.605,Z 604.191,A -85,B 0,C 180,E1 -16652.772,E2 -16652.772} C_VEL
LIN {X 0,Y 290.407,Z 603.877,A -85,B 0,C 180,E1 -16654.163,E2 -16654.163} C_VEL
LIN {X 0,Y 290.073,Z 602.275,A -85,B 0,C 180,E1 -16656.599,E2 -16656.599} C_VEL
LIN {X 0,Y 289.972,Z 599.331,A -85,B 0,C 180,E1 -16659.064,E2 -16659.064} C_VEL
LIN {X 0,Y 290.245,Z 595.752,A -85,B 0,C 180,E1 -16661.169,E2 -16661.169} C_VEL
LIN {X 0,Y 291.089,Z 591.135,A -85,B 0,C 180,E1 -16663.26,E2 -16663.26} C_VEL
LIN {X 0,Y 292.363,Z 585.386,A -85,B 0,C 180,E1 -16665.333,E2 -16665.333} C_VEL
LIN {X 0,Y 293.999,Z 578.391,A -85,B 0,C 180,E1 -16667.386,E2 -16667.386} C_VEL
LIN {X 0,Y 296.237,Z 569.937,A -85,B 0,C 180,E1 -16669.399,E2 -16669.399} C_VEL
LIN {X 0,Y 299.061,Z 559.619,A -85,B 0,C 180,E1 -16671.362,E2 -16671.362} C_VEL
LIN {X 0,Y 302.098,Z 548.192,A -85,B 0,C 180,E1 -16673.115,E2 -16673.115} C_VEL
LIN {X 0,Y 305.314,Z 535.37,A -85,B 0,C 180,E1 -16674.659,E2 -16674.659} C_VEL
LIN {X 0,Y 308.272,Z 522.661,A -85,B 0,C 180,E1 -16675.85,E2 -16675.85} C_VEL
LIN {X 0,Y 311.15,Z 507.579,A -85,B 0,C 180,E1 -16676.946,E2 -16676.946} C_VEL
LIN {X 0,Y 313.609,Z 491.64,A -85,B 0,C 180,E1 -16677.756,E2 -16677.756} C_VEL
LIN {X 0,Y 317.226,Z 454.214,A -85,B 0,C 180,E1 -16679.24,E2 -16679.24} C_VEL
LIN {X 0,Y 317.367,Z 441.245,A -85,B 0,C 180,E1 -16679.999,E2 -16679.999} C_VEL
LIN {X 0,Y 316.945,Z 429.227,A -85,B 0,C 180,E1 -16680.86,E2 -16680.86} C_VEL
LIN {X 0,Y 315.911,Z 415.333,A -85,B 0,C 180,E1 -16682.06,E2 -16682.06} C_VEL
LIN {X 0,Y 314.383,Z 401.35,A -85,B 0,C 180,E1 -16683.517,E2 -16683.517} C_VEL
LIN {X 0,Y 313.722,Z 396.855,A -85,B 0,C 180,E1 -16684.074,E2 -16684.074} C_VEL
LIN {X 0,Y 311.818,Z 391.753,A -85,B 0,C 180,E1 -16685.119,E2 -16685.119} C_VEL
LIN {X 0,Y 308.697,Z 384.27,A -85,B 0,C 180,E1 -16687.009,E2 -16687.009} C_VEL
LIN {X 0,Y 304.258,Z 374.528,A -85,B 0,C 180,E1 -16690.526,E2 -16690.526} C_VEL
LIN {X 0,Y 302.098,Z 370.077,A -85,B 0,C 180,E1 -16693.209,E2 -16693.209} C_VEL
LIN {X 0,Y 301.242,Z 367.323,A -85,B 0,C 180,E1 -16695.58,E2 -16695.58} C_VEL
LIN {X 0,Y 301.451,Z 365.339,A -85,B 0,C 180,E1 -16698.249,E2 -16698.249} C_VEL
LIN {X 0,Y 302.511,Z 365.577,A -85,B 0,C 180,E1 -16700.716,E2 -16700.716} C_VEL
LIN {X 0,Y 305.041,Z 366.309,A -85,B 0,C 180,E1 -16703.345,E2 -16703.345} C_VEL
LIN {X 0,Y 307.902,Z 368.721,A -85,B 0,C 180,E1 -16705.516,E2 -16705.516} C_VEL
LIN {X 0,Y 311.665,Z 372.739,A -85,B 0,C 180,E1 -16707.715,E2 -16707.715} C_VEL
LIN {X 0,Y 314.691,Z 376.12,A -85,B 0,C 180,E1 -16709.173,E2 -16709.173} C_VEL
LIN {X 0,Y 318.884,Z 383.342,A -85,B 0,C 180,E1 -16711.075,E2 -16711.075} C_VEL
LIN {X 0,Y 322.409,Z 390.328,A -85,B 0,C 180,E1 -16712.508,E2 -16712.508} C_VEL
LIN {X 0,Y 317.892,Z 431.056,A -85,B 0,C 180,E1 -16714.153,E2 -16714.153} C_VEL
LIN {X 0,Y 316.471,Z 448.409,A -85,B 0,C 180,E1 -16714.998,E2 -16714.998} C_VEL
LIN {X 0,Y 315.187,Z 460.454,A -85,B 0,C 180,E1 -16715.812,E2 -16715.812} C_VEL
LIN {X 0,Y 313.348,Z 472.736,A -85,B 0,C 180,E1 -16716.89,E2 -16716.89} C_VEL
LIN {X 0,Y 311.518,Z 482.808,A -85,B 0,C 180,E1 -16717.989,E2 -16717.989} C_VEL
LIN {X 0,Y 309.437,Z 492.274,A -85,B 0,C 180,E1 -16719.241,E2 -16719.241} C_VEL
LIN {X 0,Y 306.821,Z 502.641,A -85,B 0,C 180,E1 -16720.948,E2 -16720.948} C_VEL
LIN {X 0,Y 304.569,Z 510.504,A -85,B 0,C 180,E1 -16722.543,E2 -16722.543} C_VEL
LIN {X 0,Y 302.095,Z 518.215,A -85,B 0,C 180,E1 -16724.482,E2 -16724.482} C_VEL
LIN {X 0,Y 299.848,Z 524.395,A -85,B 0,C 180,E1 -16726.444,E2 -16726.444} C_VEL
LIN {X 0,Y 297.868,Z 529.276,A -85,B 0,C 180,E1 -16728.43,E2 -16728.43} C_VEL
LIN {X 0,Y 296.145,Z 533.006,A -85,B 0,C 180,E1 -16730.437,E2 -16730.437} C_VEL
LIN {X 0,Y 295.103,Z 534.929,A -85,B 0,C 180,E1 -16731.784,E2 -16731.784} C_VEL
LIN {X 0,Y 294.253,Z 536.358,A -85,B 0,C 180,E1 -16733.141,E2 -16733.141} C_VEL
LIN {X 0,Y 293.499,Z 537.343,A -85,B 0,C 180,E1 -16734.503,E2 -16734.503} C_VEL
LIN {X 0,Y 292.826,Z 537.931,A -85,B 0,C 180,E1 -16735.87,E2 -16735.87} C_VEL
LIN {X 0,Y 292.319,Z 538.091,A -85,B 0,C 180,E1 -16737.243,E2 -16737.243} C_VEL
LIN {X 0,Y 291.845,Z 537.798,A -85,B 0,C 180,E1 -16738.619,E2 -16738.619} C_VEL
LIN {X 0,Y 291.603,Z 537.08,A -85,B 0,C 180,E1 -16739.999,E2 -16739.999} C_VEL
LIN {X 0,Y 291.132,Z 535.99,A -85,B 0,C 180,E1 -16741.383,E2 -16741.383} C_VEL
LIN {X 0,Y 290.869,Z 533.47,A -85,B 0,C 180,E1 -16743.462,E2 -16743.462} C_VEL
LIN {X 0,Y 291.05,Z 529.911,A -85,B 0,C 180,E1 -16745.542,E2 -16745.542} C_VEL
LIN {X 0,Y 291.151,Z 524.522,A -85,B 0,C 180,E1 -16747.898,E2 -16747.898} C_VEL
LIN {X 0,Y 291.464,Z 518.143,A -85,B 0,C 180,E1 -16750.067,E2 -16750.067} C_VEL
LIN {X 0,Y 291.957,Z 510.497,A -85,B 0,C 180,E1 -16752.159,E2 -16752.159} C_VEL
LIN {X 0,Y 292.656,Z 500.936,A -85,B 0,C 180,E1 -16754.249,E2 -16754.249} C_VEL
LIN {X 0,Y 293.371,Z 491.186,A -85,B 0,C 180,E1 -16755.991,E2 -16755.991} C_VEL
LIN {X 0,Y 294.026,Z 480.785,A -85,B 0,C 180,E1 -16757.509,E2 -16757.509} C_VEL
LIN {X 0,Y 294.825,Z 468.58,A -85,B 0,C 180,E1 -16758.952,E2 -16758.952} C_VEL
LIN {X 0,Y 295.501,Z 455.364,A -85,B 0,C 180,E1 -16760.172,E2 -16760.172} C_VEL
LIN {X 0,Y 296.167,Z 441.643,A -85,B 0,C 180,E1 -16761.124,E2 -16761.124} C_VEL
LIN {X 0,Y 296.432,Z 427.849,A -85,B 0,C 180,E1 -16761.788,E2 -16761.788} C_VEL
LIN {X 0,Y 298.138,Z 367.027,A -85,B 0,C 180,E1 -16763.907,E2 -16763.907} C_VEL
LIN {X 0,Y 291.493,Z 345.177,A -85,B 0,C 180,E1 -16765.005,E2 -16765.005} C_VEL
LIN {X 0,Y 291.385,Z 345.191,A -85,B 0,C 180,E1 -16768.841,E2 -16768.841} C_VEL
LIN {X 0,Y 291.343,Z 345.193,A -85,B 0,C 180,E1 -16772.403,E2 -16772.403} C_VEL
LIN {X 0,Y 291.359,Z 345.19,A -85,B 0,C 180,E1 -16775.373,E2 -16775.373} C_VEL
LIN {X 0,Y 291.346,Z 345.195,A -85,B 0,C 180,E1 -16778.842,E2 -16778.842} C_VEL
LIN {X 0,Y 291.318,Z 345.197,A -85,B 0,C 180,E1 -16782.492,E2 -16782.492} C_VEL
LIN {X 0,Y 291.317,Z 345.196,A -85,B 0,C 180,E1 -16786.364,E2 -16786.364} C_VEL
LIN {X 0,Y 291.385,Z 345.189,A -85,B 0,C 180,E1 -16790.516,E2 -16790.516} C_VEL
LIN {X 0,Y 291.423,Z 345.184,A -85,B 0,C 180,E1 -16792.922,E2 -16792.922} C_VEL
LIN {X 0,Y 291.342,Z 345.192,A -85,B 0,C 180,E1 -16796.301,E2 -16796.301} C_VEL
LIN {X 0,Y 291.381,Z 345.189,A -85,B 0,C 180,E1 -16800.261,E2 -16800.261} C_VEL
LIN {X 0,Y 291.41,Z 345.184,A -85,B 0,C 180,E1 -16804.271,E2 -16804.271} C_VEL
LIN {X 0,Y 291.379,Z 345.187,A -85,B 0,C 180,E1 -16807.299,E2 -16807.299} C_VEL
LIN {X 0,Y 291.455,Z 345.18,A -85,B 0,C 180,E1 -16810.27,E2 -16810.27} C_VEL
LIN {X 0,Y 291.552,Z 345.169,A -85,B 0,C 180,E1 -16814.624,E2 -16814.624} C_VEL
LIN {X 0,Y 291.534,Z 345.169,A -85,B 0,C 180,E1 -16818.881,E2 -16818.881} C_VEL
LIN {X 0,Y 291.706,Z 345.145,A -85,B 0,C 180,E1 -16821.689,E2 -16821.689} C_VEL
LIN {X 0,Y 291.628,Z 345.161,A -85,B 0,C 180,E1 -16824.468,E2 -16824.468} C_VEL
LIN {X 0,Y 291.887,Z 345.126,A -85,B 0,C 180,E1 -16828.621,E2 -16828.621} C_VEL
LIN {X 0,Y 291.887,Z 345.123,A -85,B 0,C 180,E1 -16831.38,E2 -16831.38} C_VEL
LIN {X 0,Y 291.744,Z 345.142,A -85,B 0,C 180,E1 -16836.918,E2 -16836.918} C_VEL
LIN {X 0,Y 291.627,Z 345.156,A -85,B 0,C 180,E1 -16839.712,E2 -16839.712} C_VEL
LIN {X 0,Y 291.52,Z 345.172,A -85,B 0,C 180,E1 -16843.951,E2 -16843.951} C_VEL
LIN {X 0,Y 291.485,Z 345.174,A -85,B 0,C 180,E1 -16846.818,E2 -16846.818} C_VEL
LIN {X 0,Y 291.448,Z 345.18,A -85,B 0,C 180,E1 -16849.875,E2 -16849.875} C_VEL
LIN {X 0,Y 291.398,Z 345.189,A -85,B 0,C 180,E1 -16854.206,E2 -16854.206} C_VEL
LIN {X 0,Y 291.419,Z 345.181,A -85,B 0,C 180,E1 -16857.272,E2 -16857.272} C_VEL
LIN {X 0,Y 291.333,Z 345.195,A -85,B 0,C 180,E1 -16860.438,E2 -16860.438} C_VEL
LIN {X 0,Y 291.343,Z 345.192,A -85,B 0,C 180,E1 -16863.699,E2 -16863.699} C_VEL
LIN {X 0,Y 291.393,Z 345.185,A -85,B 0,C 180,E1 -16867.259,E2 -16867.259} C_VEL
LIN {X 0,Y 291.333,Z 345.193,A -85,B 0,C 180,E1 -16870.643,E2 -16870.643} C_VEL
LIN {X 0,Y 291.29,Z 345.2,A -85,B 0,C 180,E1 -16874.403,E2 -16874.403} C_VEL
LIN {X 0,Y 291.326,Z 345.195,A -85,B 0,C 180,E1 -16878.405,E2 -16878.405} C_VEL
LIN {X 0,Y 291.364,Z 345.188,A -85,B 0,C 180,E1 -16881.161,E2 -16881.161} C_VEL
LIN {X 0,Y 291.363,Z 345.189,A -85,B 0,C 180,E1 -16884.627,E2 -16884.627} C_VEL
LIN {X 0,Y 291.404,Z 345.266,A -85,B 0,C 180,E1 -16888.741,E2 -16888.741} C_VEL
LIN {X 0,Y 298.686,Z 367.788,A -85,B 0,C 180,E1 -16889.878,E2 -16889.878} C_VEL
LIN {X 0,Y 296.855,Z 430.879,A -85,B 0,C 180,E1 -16891.98,E2 -16891.98} C_VEL
LIN {X 0,Y 296.574,Z 444.269,A -85,B 0,C 180,E1 -16892.669,E2 -16892.669} C_VEL
LIN {X 0,Y 295.808,Z 458.809,A -85,B 0,C 180,E1 -16893.737,E2 -16893.737} C_VEL
LIN {X 0,Y 295.14,Z 470.816,A -85,B 0,C 180,E1 -16894.916,E2 -16894.916} C_VEL
LIN {X 0,Y 294.28,Z 482.977,A -85,B 0,C 180,E1 -16896.421,E2 -16896.421} C_VEL
LIN {X 0,Y 293.427,Z 493.344,A -85,B 0,C 180,E1 -16898.023,E2 -16898.023} C_VEL
LIN {X 0,Y 292.723,Z 502.941,A -85,B 0,C 180,E1 -16899.835,E2 -16899.835} C_VEL
LIN {X 0,Y 292.605,Z 504.276,A -85,B 0,C 180,E1 -16900.116,E2 -16900.116} C_VEL
LIN {X 0,Y 291.53,Z 508.169,A -85,B 0,C 180,E1 -16900.975,E2 -16900.975} C_VEL
LIN {X 0,Y 286.817,Z 516.299,A -85,B 0,C 180,E1 -16903,E2 -16903} C_VEL
LIN {X 0,Y 284.668,Z 520.521,A -85,B 0,C 180,E1 -16904.272,E2 -16904.272} C_VEL
LIN {X 0,Y 284.253,Z 522.474,A -85,B 0,C 180,E1 -16904.952,E2 -16904.952} C_VEL
LIN {X 0,Y 283.959,Z 527.848,A -85,B 0,C 180,E1 -16907.13,E2 -16907.13} C_VEL
LIN {X 0,Y 283.913,Z 531.955,A -85,B 0,C 180,E1 -16909.301,E2 -16909.301} C_VEL
LIN {X 0,Y 284.107,Z 535.174,A -85,B 0,C 180,E1 -16911.688,E2 -16911.688} C_VEL
LIN {X 0,Y 284.44,Z 537.331,A -85,B 0,C 180,E1 -16914.329,E2 -16914.329} C_VEL
LIN {X 0,Y 284.757,Z 537.9,A -85,B 0,C 180,E1 -16915.754,E2 -16915.754} C_VEL
LIN {X 0,Y 285.265,Z 537.979,A -85,B 0,C 180,E1 -16917.176,E2 -16917.176} C_VEL
LIN {X 0,Y 285.821,Z 537.657,A -85,B 0,C 180,E1 -16918.592,E2 -16918.592} C_VEL
LIN {X 0,Y 286.497,Z 536.93,A -85,B 0,C 180,E1 -16920.001,E2 -16920.001} C_VEL
LIN {X 0,Y 287.29,Z 535.729,A -85,B 0,C 180,E1 -16921.402,E2 -16921.402} C_VEL
LIN {X 0,Y 288.687,Z 533.122,A -85,B 0,C 180,E1 -16923.491,E2 -16923.491} C_VEL
LIN {X 0,Y 290.351,Z 529.441,A -85,B 0,C 180,E1 -16925.557,E2 -16925.557} C_VEL
LIN {X 0,Y 292.255,Z 524.598,A -85,B 0,C 180,E1 -16927.601,E2 -16927.601} C_VEL
LIN {X 0,Y 294.48,Z 518.503,A -85,B 0,C 180,E1 -16929.618,E2 -16929.618} C_VEL
LIN {X 0,Y 296.904,Z 510.865,A -85,B 0,C 180,E1 -16931.608,E2 -16931.608} C_VEL
LIN {X 0,Y 299.079,Z 503.06,A -85,B 0,C 180,E1 -16933.246,E2 -16933.246} C_VEL
LIN {X 0,Y 301.699,Z 492.606,A -85,B 0,C 180,E1 -16935.021,E2 -16935.021} C_VEL
LIN {X 0,Y 303.956,Z 481.98,A -85,B 0,C 180,E1 -16936.454,E2 -16936.454} C_VEL
LIN {X 0,Y 306.042,Z 470.154,A -85,B 0,C 180,E1 -16937.715,E2 -16937.715} C_VEL
LIN {X 0,Y 307.794,Z 456.791,A -85,B 0,C 180,E1 -16938.816,E2 -16938.816} C_VEL
LIN {X 0,Y 308.987,Z 443.321,A -85,B 0,C 180,E1 -16939.646,E2 -16939.646} C_VEL
LIN {X 0,Y 311.095,Z 416.642,A -85,B 0,C 180,E1 -16940.755,E2 -16940.755} C_VEL
LIN {X 0,Y 313.682,Z 389.698,A -85,B 0,C 180,E1 -16941.791,E2 -16941.791} C_VEL
LIN {X 0,Y 309.668,Z 382.067,A -85,B 0,C 180,E1 -16943.251,E2 -16943.251} C_VEL
LIN {X 0,Y 305.316,Z 374.786,A -85,B 0,C 180,E1 -16944.976,E2 -16944.976} C_VEL
LIN {X 0,Y 302.851,Z 370.99,A -85,B 0,C 180,E1 -16946.063,E2 -16946.063} C_VEL
LIN {X 0,Y 300.384,Z 367.257,A -85,B 0,C 180,E1 -16947.242,E2 -16947.242} C_VEL
LIN {X 0,Y 298.004,Z 363.953,A -85,B 0,C 180,E1 -16948.512,E2 -16948.512} C_VEL
LIN {X 0,Y 297.24,Z 362.644,A -85,B 0,C 180,E1 -16948.974,E2 -16948.974} C_VEL
LIN {X 0,Y 294.883,Z 360.148,A -85,B 0,C 180,E1 -16950.409,E2 -16950.409} C_VEL
LIN {X 0,Y 293.752,Z 357.657,A -85,B 0,C 180,E1 -16951.383,E2 -16951.383} C_VEL
LIN {X 0,Y 290.878,Z 355.325,A -85,B 0,C 180,E1 -16953.76,E2 -16953.76} C_VEL
LIN {X 0,Y 289.87,Z 353.671,A -85,B 0,C 180,E1 -16955.085,E2 -16955.085} C_VEL
LIN {X 0,Y 288.512,Z 352.365,A -85,B 0,C 180,E1 -16957.517,E2 -16957.517} C_VEL
LIN {X 0,Y 287.993,Z 352.416,A -85,B 0,C 180,E1 -16960.076,E2 -16960.076} C_VEL
LIN {X 0,Y 288.876,Z 354.242,A -85,B 0,C 180,E1 -16963.124,E2 -16963.124} C_VEL
LIN {X 0,Y 291.349,Z 356.936,A -85,B 0,C 180,E1 -16966.359,E2 -16966.359} C_VEL
LIN {X 0,Y 293.167,Z 360.376,A -85,B 0,C 180,E1 -16968.399,E2 -16968.399} C_VEL
LIN {X 0,Y 295.14,Z 362.903,A -85,B 0,C 180,E1 -16969.803,E2 -16969.803} C_VEL
LIN {X 0,Y 298.752,Z 367.983,A -85,B 0,C 180,E1 -16971.952,E2 -16971.952} C_VEL
LIN {X 0,Y 300.443,Z 370.905,A -85,B 0,C 180,E1 -16972.879,E2 -16972.879} C_VEL
LIN {X 0,Y 304.71,Z 384.867,A -85,B 0,C 180,E1 -16975.38,E2 -16975.38} C_VEL
LIN {X 0,Y 305.881,Z 390.073,A -85,B 0,C 180,E1 -16976.089,E2 -16976.089} C_VEL
LIN {X 0,Y 307.1,Z 405.82,A -85,B 0,C 180,E1 -16977.478,E2 -16977.478} C_VEL
LIN {X 0,Y 308.158,Z 426.727,A -85,B 0,C 180,E1 -16979.043,E2 -16979.043} C_VEL
LIN {X 0,Y 308.633,Z 444.176,A -85,B 0,C 180,E1 -16980.168,E2 -16980.168} C_VEL
LIN {X 0,Y 308.482,Z 457.892,A -85,B 0,C 180,E1 -16980.904,E2 -16980.904} C_VEL
LIN {X 0,Y 305.086,Z 495.059,A -85,B 0,C 180,E1 -16982.333,E2 -16982.333} C_VEL
LIN {X 0,Y 303.233,Z 508.105,A -85,B 0,C 180,E1 -16983.038,E2 -16983.038} C_VEL
LIN {X 0,Y 300.674,Z 521.649,A -85,B 0,C 180,E1 -16984.006,E2 -16984.006} C_VEL
LIN {X 0,Y 297.777,Z 534.686,A -85,B 0,C 180,E1 -16985.233,E2 -16985.233} C_VEL
LIN {X 0,Y 294.873,Z 546.376,A -85,B 0,C 180,E1 -16986.656,E2 -16986.656} C_VEL
LIN {X 0,Y 292.373,Z 556.094,A -85,B 0,C 180,E1 -16988.124,E2 -16988.124} C_VEL
LIN {X 0,Y 289.913,Z 565.212,A -85,B 0,C 180,E1 -16989.791,E2 -16989.791} C_VEL
LIN {X 0,Y 287.453,Z 574.217,A -85,B 0,C 180,E1 -16991.836,E2 -16991.836} C_VEL
LIN {X 0,Y 285.839,Z 580.975,A -85,B 0,C 180,E1 -16993.721,E2 -16993.721} C_VEL
LIN {X 0,Y 284.458,Z 586.832,A -85,B 0,C 180,E1 -16995.696,E2 -16995.696} C_VEL
LIN {X 0,Y 283.539,Z 591.926,A -85,B 0,C 180,E1 -16997.837,E2 -16997.837} C_VEL
LIN {X 0,Y 283.042,Z 595.93,A -85,B 0,C 180,E1 -16999.99,E2 -16999.99} C_VEL
LIN {X 0,Y 282.914,Z 598.041,A -85,B 0,C 180,E1 -17001.428,E2 -17001.428} C_VEL
LIN {X 0,Y 283.06,Z 600.113,A -85,B 0,C 180,E1 -17003.293,E2 -17003.293} C_VEL
LIN {X 0,Y 283.414,Z 601.726,A -85,B 0,C 180,E1 -17005.733,E2 -17005.733} C_VEL
LIN {X 0,Y 283.631,Z 602.075,A -85,B 0,C 180,E1 -17007.159,E2 -17007.159} C_VEL
LIN {X 0,Y 284.064,Z 601.763,A -85,B 0,C 180,E1 -17009.468,E2 -17009.468} C_VEL
LIN {X 0,Y 283.783,Z 602.869,A -85,B 0,C 180,E1 -17011.419,E2 -17011.419} C_VEL
LIN {X 0,Y 283.563,Z 603.122,A -85,B 0,C 180,E1 -17012.841,E2 -17012.841} C_VEL
LIN {X 0,Y 283.339,Z 602.928,A -85,B 0,C 180,E1 -17014.267,E2 -17014.267} C_VEL
LIN {X 0,Y 282.996,Z 601.63,A -85,B 0,C 180,E1 -17016.596,E2 -17016.596} C_VEL
LIN {X 0,Y 282.882,Z 599.626,A -85,B 0,C 180,E1 -17018.573,E2 -17018.573} C_VEL
LIN {X 0,Y 283.072,Z 596.536,A -85,B 0,C 180,E1 -17020.731,E2 -17020.731} C_VEL
LIN {X 0,Y 283.8,Z 592.455,A -85,B 0,C 180,E1 -17022.878,E2 -17022.878} C_VEL
LIN {X 0,Y 284.939,Z 587.312,A -85,B 0,C 180,E1 -17025.009,E2 -17025.009} C_VEL
LIN {X 0,Y 286.881,Z 579.831,A -85,B 0,C 180,E1 -17027.463,E2 -17027.463} C_VEL
LIN {X 0,Y 289.125,Z 571.937,A -85,B 0,C 180,E1 -17029.526,E2 -17029.526} C_VEL
LIN {X 0,Y 292.016,Z 562.361,A -85,B 0,C 180,E1 -17031.532,E2 -17031.532} C_VEL
LIN {X 0,Y 295.081,Z 551.836,A -85,B 0,C 180,E1 -17033.326,E2 -17033.326} C_VEL
LIN {X 0,Y 298.285,Z 540.205,A -85,B 0,C 180,E1 -17034.908,E2 -17034.908} C_VEL
LIN {X 0,Y 301.67,Z 527.398,A -85,B 0,C 180,E1 -17036.273,E2 -17036.273} C_VEL
LIN {X 0,Y 304.822,Z 513.123,A -85,B 0,C 180,E1 -17037.459,E2 -17037.459} C_VEL
LIN {X 0,Y 307.426,Z 499.218,A -85,B 0,C 180,E1 -17038.318,E2 -17038.318} C_VEL
LIN {X 0,Y 309.521,Z 483.69,A -85,B 0,C 180,E1 -17039.03,E2 -17039.03} C_VEL
LIN {X 0,Y 312.453,Z 454.785,A -85,B 0,C 180,E1 -17040.209,E2 -17040.209} C_VEL
LIN {X 0,Y 312.725,Z 442.724,A -85,B 0,C 180,E1 -17040.941,E2 -17040.941} C_VEL
LIN {X 0,Y 312.409,Z 429.661,A -85,B 0,C 180,E1 -17041.924,E2 -17041.924} C_VEL
LIN {X 0,Y 311.543,Z 415.759,A -85,B 0,C 180,E1 -17043.197,E2 -17043.197} C_VEL
LIN {X 0,Y 310.216,Z 401.798,A -85,B 0,C 180,E1 -17044.761,E2 -17044.761} C_VEL
LIN {X 0,Y 308.623,Z 397.182,A -85,B 0,C 180,E1 -17045.732,E2 -17045.732} C_VEL
LIN {X 0,Y 305.892,Z 390.121,A -85,B 0,C 180,E1 -17047.553,E2 -17047.553} C_VEL
LIN {X 0,Y 301.998,Z 380.807,A -85,B 0,C 180,E1 -17050.985,E2 -17050.985} C_VEL
LIN {X 0,Y 300.019,Z 376.227,A -85,B 0,C 180,E1 -17053.865,E2 -17053.865} C_VEL
LIN {X 0,Y 299.454,Z 373.317,A -85,B 0,C 180,E1 -17056.682,E2 -17056.682} C_VEL
LIN {X 0,Y 299.829,Z 372.202,A -85,B 0,C 180,E1 -17058.597,E2 -17058.597} C_VEL
LIN {X 0,Y 301.484,Z 372.645,A -85,B 0,C 180,E1 -17061.608,E2 -17061.608} C_VEL
LIN {X 0,Y 303.146,Z 373.13,A -85,B 0,C 180,E1 -17063.21,E2 -17063.21} C_VEL
LIN {X 0,Y 306.336,Z 376.077,A -85,B 0,C 180,E1 -17065.682,E2 -17065.682} C_VEL
LIN {X 0,Y 309.415,Z 379.473,A -85,B 0,C 180,E1 -17067.523,E2 -17067.523} C_VEL
LIN {X 0,Y 311.938,Z 382.351,A -85,B 0,C 180,E1 -17068.788,E2 -17068.788} C_VEL
LIN {X 0,Y 315.701,Z 389.261,A -85,B 0,C 180,E1 -17070.624,E2 -17070.624} C_VEL
LIN {X 0,Y 317.888,Z 393.606,A -85,B 0,C 180,E1 -17071.583,E2 -17071.583} C_VEL
LIN {X 0,Y 313.137,Z 433.741,A -85,B 0,C 180,E1 -17073.259,E2 -17073.259} C_VEL
LIN {X 0,Y 311.612,Z 450.779,A -85,B 0,C 180,E1 -17074.133,E2 -17074.133} C_VEL
LIN {X 0,Y 309.897,Z 464.357,A -85,B 0,C 180,E1 -17075.113,E2 -17075.113} C_VEL
LIN {X 0,Y 307.758,Z 476.834,A -85,B 0,C 180,E1 -17076.284,E2 -17076.284} C_VEL
LIN {X 0,Y 305.274,Z 488.675,A -85,B 0,C 180,E1 -17077.711,E2 -17077.711} C_VEL
LIN {X 0,Y 302.644,Z 498.978,A -85,B 0,C 180,E1 -17079.259,E2 -17079.259} C_VEL
LIN {X 0,Y 299.66,Z 509.168,A -85,B 0,C 180,E1 -17081.186,E2 -17081.186} C_VEL
LIN {X 0,Y 296.918,Z 517.302,A -85,B 0,C 180,E1 -17083.144,E2 -17083.144} C_VEL
LIN {X 0,Y 294.816,Z 522.886,A -85,B 0,C 180,E1 -17084.797,E2 -17084.797} C_VEL
LIN {X 0,Y 292.536,Z 528.308,A -85,B 0,C 180,E1 -17086.806,E2 -17086.806} C_VEL
LIN {X 0,Y 290.533,Z 532.544,A -85,B 0,C 180,E1 -17088.841,E2 -17088.841} C_VEL
LIN {X 0,Y 289.368,Z 534.762,A -85,B 0,C 180,E1 -17090.211,E2 -17090.211} C_VEL
LIN {X 0,Y 288.274,Z 536.504,A -85,B 0,C 180,E1 -17091.588,E2 -17091.588} C_VEL
LIN {X 0,Y 287.348,Z 537.791,A -85,B 0,C 180,E1 -17092.975,E2 -17092.975} C_VEL
LIN {X 0,Y 286.57,Z 538.661,A -85,B 0,C 180,E1 -17094.37,E2 -17094.37} C_VEL
LIN {X 0,Y 285.848,Z 539.112,A -85,B 0,C 180,E1 -17095.769,E2 -17095.769} C_VEL
LIN {X 0,Y 285.314,Z 539.104,A -85,B 0,C 180,E1 -17097.176,E2 -17097.176} C_VEL
LIN {X 0,Y 284.822,Z 538.699,A -85,B 0,C 180,E1 -17098.585,E2 -17098.585} C_VEL
LIN {X 0,Y 284.547,Z 537.874,A -85,B 0,C 180,E1 -17099.999,E2 -17099.999} C_VEL
LIN {X 0,Y 284.052,Z 536.612,A -85,B 0,C 180,E1 -17101.417,E2 -17101.417} C_VEL
LIN {X 0,Y 283.794,Z 533.89,A -85,B 0,C 180,E1 -17103.549,E2 -17103.549} C_VEL
LIN {X 0,Y 283.967,Z 530.113,A -85,B 0,C 180,E1 -17105.681,E2 -17105.681} C_VEL
LIN {X 0,Y 284.062,Z 524.958,A -85,B 0,C 180,E1 -17107.912,E2 -17107.912} C_VEL
LIN {X 0,Y 284.42,Z 517.849,A -85,B 0,C 180,E1 -17110.319,E2 -17110.319} C_VEL
LIN {X 0,Y 284.942,Z 509.826,A -85,B 0,C 180,E1 -17112.463,E2 -17112.463} C_VEL
LIN {X 0,Y 285.681,Z 499.922,A -85,B 0,C 180,E1 -17114.605,E2 -17114.605} C_VEL
LIN {X 0,Y 286.468,Z 488.698,A -85,B 0,C 180,E1 -17116.544,E2 -17116.544} C_VEL
LIN {X 0,Y 287.239,Z 476.956,A -85,B 0,C 180,E1 -17118.177,E2 -17118.177} C_VEL
LIN {X 0,Y 288.075,Z 464.059,A -85,B 0,C 180,E1 -17119.599,E2 -17119.599} C_VEL
LIN {X 0,Y 288.711,Z 451.493,A -85,B 0,C 180,E1 -17120.668,E2 -17120.668} C_VEL
LIN {X 0,Y 289.25,Z 437.402,A -85,B 0,C 180,E1 -17121.561,E2 -17121.561} C_VEL
LIN {X 0,Y 289.533,Z 421.071,A -85,B 0,C 180,E1 -17122.241,E2 -17122.241} C_VEL
LIN {X 0,Y 291.203,Z 368.454,A -85,B 0,C 180,E1 -17124.134,E2 -17124.134} C_VEL
LIN {X 0,Y 284.434,Z 346.054,A -85,B 0,C 180,E1 -17125.294,E2 -17125.294} C_VEL
LIN {X 0,Y 284.359,Z 346.06,A -85,B 0,C 180,E1 -17129.623,E2 -17129.623} C_VEL
LIN {X 0,Y 284.305,Z 346.072,A -85,B 0,C 180,E1 -17132.944,E2 -17132.944} C_VEL
LIN {X 0,Y 284.329,Z 346.067,A -85,B 0,C 180,E1 -17136.386,E2 -17136.386} C_VEL
LIN {X 0,Y 284.304,Z 346.068,A -85,B 0,C 180,E1 -17139.994,E2 -17139.994} C_VEL
LIN {X 0,Y 284.264,Z 346.074,A -85,B 0,C 180,E1 -17144.194,E2 -17144.194} C_VEL
LIN {X 0,Y 284.27,Z 346.072,A -85,B 0,C 180,E1 -17148.124,E2 -17148.124} C_VEL
LIN {X 0,Y 284.333,Z 346.066,A -85,B 0,C 180,E1 -17152.274,E2 -17152.274} C_VEL
LIN {X 0,Y 284.321,Z 346.065,A -85,B 0,C 180,E1 -17155.352,E2 -17155.352} C_VEL
LIN {X 0,Y 284.291,Z 346.074,A -85,B 0,C 180,E1 -17158.725,E2 -17158.725} C_VEL
LIN {X 0,Y 284.391,Z 346.059,A -85,B 0,C 180,E1 -17162.827,E2 -17162.827} C_VEL
LIN {X 0,Y 284.364,Z 346.065,A -85,B 0,C 180,E1 -17166.707,E2 -17166.707} C_VEL
LIN {X 0,Y 284.4,Z 346.056,A -85,B 0,C 180,E1 -17171.262,E2 -17171.262} C_VEL
LIN {X 0,Y 284.489,Z 346.049,A -85,B 0,C 180,E1 -17174.459,E2 -17174.459} C_VEL
LIN {X 0,Y 284.486,Z 346.049,A -85,B 0,C 180,E1 -17178.602,E2 -17178.602} C_VEL
LIN {X 0,Y 284.656,Z 346.023,A -85,B 0,C 180,E1 -17181.481,E2 -17181.481} C_VEL
LIN {X 0,Y 284.599,Z 346.035,A -85,B 0,C 180,E1 -17184.331,E2 -17184.331} C_VEL
LIN {X 0,Y 284.853,Z 346.002,A -85,B 0,C 180,E1 -17188.586,E2 -17188.586} C_VEL
LIN {X 0,Y 284.853,Z 345.999,A -85,B 0,C 180,E1 -17191.414,E2 -17191.414} C_VEL
LIN {X 0,Y 284.696,Z 346.019,A -85,B 0,C 180,E1 -17197.09,E2 -17197.09} C_VEL
LIN {X 0,Y 284.564,Z 346.037,A -85,B 0,C 180,E1 -17199.956,E2 -17199.956} C_VEL
LIN {X 0,Y 284.479,Z 346.051,A -85,B 0,C 180,E1 -17204.303,E2 -17204.303} C_VEL
LIN {X 0,Y 284.423,Z 346.052,A -85,B 0,C 180,E1 -17207.249,E2 -17207.249} C_VEL
LIN {X 0,Y 284.377,Z 346.064,A -85,B 0,C 180,E1 -17210.243,E2 -17210.243} C_VEL
LIN {X 0,Y 284.367,Z 346.062,A -85,B 0,C 180,E1 -17213.876,E2 -17213.876} C_VEL
LIN {X 0,Y 284.394,Z 346.056,A -85,B 0,C 180,E1 -17217.174,E2 -17217.174} C_VEL
LIN {X 0,Y 284.293,Z 346.069,A -85,B 0,C 180,E1 -17221.275,E2 -17221.275} C_VEL
LIN {X 0,Y 284.36,Z 346.061,A -85,B 0,C 180,E1 -17225.355,E2 -17225.355} C_VEL
LIN {X 0,Y 284.322,Z 346.07,A -85,B 0,C 180,E1 -17228.168,E2 -17228.168} C_VEL
LIN {X 0,Y 284.269,Z 346.076,A -85,B 0,C 180,E1 -17232.125,E2 -17232.125} C_VEL
LIN {X 0,Y 284.255,Z 346.078,A -85,B 0,C 180,E1 -17236.19,E2 -17236.19} C_VEL
LIN {X 0,Y 284.307,Z 346.072,A -85,B 0,C 180,E1 -17240.025,E2 -17240.025} C_VEL
LIN {X 0,Y 284.337,Z 346.066,A -85,B 0,C 180,E1 -17243.616,E2 -17243.616} C_VEL
LIN {X 0,Y 284.347,Z 346.065,A -85,B 0,C 180,E1 -17248.396,E2 -17248.396} C_VEL
LIN {X 0,Y 291.742,Z 369.177,A -85,B 0,C 180,E1 -17249.611,E2 -17249.611} C_VEL
LIN {X 0,Y 289.868,Z 430.813,A -85,B 0,C 180,E1 -17251.736,E2 -17251.736} C_VEL
LIN {X 0,Y 289.583,Z 444.4,A -85,B 0,C 180,E1 -17252.444,E2 -17252.444} C_VEL
LIN {X 0,Y 288.868,Z 457.987,A -85,B 0,C 180,E1 -17253.446,E2 -17253.446} C_VEL
LIN {X 0,Y 288.241,Z 469.599,A -85,B 0,C 180,E1 -17254.564,E2 -17254.564} C_VEL
LIN {X 0,Y 287.387,Z 481.472,A -85,B 0,C 180,E1 -17256.012,E2 -17256.012} C_VEL
LIN {X 0,Y 286.51,Z 492.36,A -85,B 0,C 180,E1 -17257.654,E2 -17257.654} C_VEL
LIN {X 0,Y 285.715,Z 502.549,A -85,B 0,C 180,E1 -17259.563,E2 -17259.563} C_VEL
LIN {X 0,Y 284.976,Z 511.712,A -85,B 0,C 180,E1 -17261.674,E2 -17261.674} C_VEL
LIN {X 0,Y 284.442,Z 519.277,A -85,B 0,C 180,E1 -17263.862,E2 -17263.862} C_VEL
LIN {X 0,Y 284.253,Z 522.474,A -85,B 0,C 180,E1 -17264.952,E2 -17264.952} C_VEL
LIN {X 0,Y 283.446,Z 525.297,A -85,B 0,C 180,E1 -17265.988,E2 -17265.988} C_VEL
LIN {X 0,Y 280.428,Z 529.454,A -85,B 0,C 180,E1 -17267.714,E2 -17267.714} C_VEL
LIN {X 0,Y 277.973,Z 532.261,A -85,B 0,C 180,E1 -17269.16,E2 -17269.16} C_VEL
LIN {X 0,Y 276.971,Z 534.052,A -85,B 0,C 180,E1 -17270.31,E2 -17270.31} C_VEL
LIN {X 0,Y 276.915,Z 534.58,A -85,B 0,C 180,E1 -17270.704,E2 -17270.704} C_VEL
LIN {X 0,Y 277.153,Z 536.89,A -85,B 0,C 180,E1 -17272.717,E2 -17272.717} C_VEL
LIN {X 0,Y 277.367,Z 538.026,A -85,B 0,C 180,E1 -17274.184,E2 -17274.184} C_VEL
LIN {X 0,Y 277.675,Z 538.737,A -85,B 0,C 180,E1 -17275.646,E2 -17275.646} C_VEL
LIN {X 0,Y 278.207,Z 539.03,A -85,B 0,C 180,E1 -17277.105,E2 -17277.105} C_VEL
LIN {X 0,Y 278.793,Z 538.869,A -85,B 0,C 180,E1 -17278.556,E2 -17278.556} C_VEL
LIN {X 0,Y 279.489,Z 538.277,A -85,B 0,C 180,E1 -17280.001,E2 -17280.001} C_VEL
LIN {X 0,Y 280.322,Z 537.279,A -85,B 0,C 180,E1 -17281.437,E2 -17281.437} C_VEL
LIN {X 0,Y 281.602,Z 535.221,A -85,B 0,C 180,E1 -17283.344,E2 -17283.344} C_VEL
LIN {X 0,Y 283.526,Z 531.556,A -85,B 0,C 180,E1 -17285.691,E2 -17285.691} C_VEL
LIN {X 0,Y 285.504,Z 527.078,A -85,B 0,C 180,E1 -17287.782,E2 -17287.782} C_VEL
LIN {X 0,Y 287.802,Z 521.294,A -85,B 0,C 180,E1 -17289.843,E2 -17289.843} C_VEL
LIN {X 0,Y 290.321,Z 514.08,A -85,B 0,C 180,E1 -17291.875,E2 -17291.875} C_VEL
LIN {X 0,Y 292.616,Z 506.828,A -85,B 0,C 180,E1 -17293.544,E2 -17293.544} C_VEL
LIN {X 0,Y 295.193,Z 497.967,A -85,B 0,C 180,E1 -17295.183,E2 -17295.183} C_VEL
LIN {X 0,Y 297.755,Z 487.121,A -85,B 0,C 180,E1 -17296.807,E2 -17296.807} C_VEL
LIN {X 0,Y 300.227,Z 474.915,A -85,B 0,C 180,E1 -17298.246,E2 -17298.246} C_VEL
LIN {X 0,Y 302.287,Z 461.896,A -85,B 0,C 180,E1 -17299.437,E2 -17299.437} C_VEL
LIN {X 0,Y 303.816,Z 447.98,A -85,B 0,C 180,E1 -17300.387,E2 -17300.387} C_VEL
LIN {X 0,Y 305.188,Z 430.226,A -85,B 0,C 180,E1 -17301.211,E2 -17301.211} C_VEL
LIN {X 0,Y 309.03,Z 393.007,A -85,B 0,C 180,E1 -17302.685,E2 -17302.685} C_VEL
LIN {X 0,Y 304.416,Z 384.27,A -85,B 0,C 180,E1 -17304.524,E2 -17304.524} C_VEL
LIN {X 0,Y 300.304,Z 377.458,A -85,B 0,C 180,E1 -17306.366,E2 -17306.366} C_VEL
LIN {X 0,Y 297.568,Z 373.285,A -85,B 0,C 180,E1 -17307.761,E2 -17307.761} C_VEL
LIN {X 0,Y 295.286,Z 369.829,A -85,B 0,C 180,E1 -17309.072,E2 -17309.072} C_VEL
LIN {X 0,Y 294.333,Z 368.637,A -85,B 0,C 180,E1 -17309.664,E2 -17309.664} C_VEL
LIN {X 0,Y 292.245,Z 365.902,A -85,B 0,C 180,E1 -17311.105,E2 -17311.105} C_VEL
LIN {X 0,Y 291.443,Z 364.237,A -85,B 0,C 180,E1 -17311.834,E2 -17311.834} C_VEL
LIN {X 0,Y 288.697,Z 361.565,A -85,B 0,C 180,E1 -17314.399,E2 -17314.399} C_VEL
LIN {X 0,Y 288.102,Z 360.459,A -85,B 0,C 180,E1 -17315.332,E2 -17315.332} C_VEL
LIN {X 0,Y 286.835,Z 359.227,A -85,B 0,C 180,E1 -17317.775,E2 -17317.775} C_VEL
LIN {X 0,Y 286.411,Z 359.495,A -85,B 0,C 180,E1 -17320.475,E2 -17320.475} C_VEL
LIN {X 0,Y 287.684,Z 362.043,A -85,B 0,C 180,E1 -17324.348,E2 -17324.348} C_VEL
LIN {X 0,Y 289.192,Z 363.789,A -85,B 0,C 180,E1 -17326.207,E2 -17326.207} C_VEL
LIN {X 0,Y 292.933,Z 369.443,A -85,B 0,C 180,E1 -17329.484,E2 -17329.484} C_VEL
LIN {X 0,Y 296.421,Z 374.6,A -85,B 0,C 180,E1 -17331.664,E2 -17331.664} C_VEL
LIN {X 0,Y 297.426,Z 376.527,A -85,B 0,C 180,E1 -17332.248,E2 -17332.248} C_VEL
LIN {X 0,Y 301.009,Z 389.495,A -85,B 0,C 180,E1 -17334.627,E2 -17334.627} C_VEL
LIN {X 0,Y 301.835,Z 393.781,A -85,B 0,C 180,E1 -17335.216,E2 -17335.216} C_VEL
LIN {X 0,Y 302.76,Z 408.843,A -85,B 0,C 180,E1 -17336.582,E2 -17336.582} C_VEL
LIN {X 0,Y 303.623,Z 431.271,A -85,B 0,C 180,E1 -17338.302,E2 -17338.302} C_VEL
LIN {X 0,Y 303.763,Z 447.953,A -85,B 0,C 180,E1 -17339.375,E2 -17339.375} C_VEL
LIN {X 0,Y 303.535,Z 458.895,A -85,B 0,C 180,E1 -17339.972,E2 -17339.972} C_VEL
LIN {X 0,Y 299.954,Z 494.503,A -85,B 0,C 180,E1 -17341.389,E2 -17341.389} C_VEL
LIN {X 0,Y 298.086,Z 506.786,A -85,B 0,C 180,E1 -17342.056,E2 -17342.056} C_VEL
LIN {X 0,Y 295.221,Z 521.121,A -85,B 0,C 180,E1 -17343.107,E2 -17343.107} C_VEL
LIN {X 0,Y 292.167,Z 533.861,A -85,B 0,C 180,E1 -17344.342,E2 -17344.342} C_VEL
LIN {X 0,Y 288.763,Z 546.674,A -85,B 0,C 180,E1 -17345.941,E2 -17345.941} C_VEL
LIN {X 0,Y 285.874,Z 557.052,A -85,B 0,C 180,E1 -17347.601,E2 -17347.601} C_VEL
LIN {X 0,Y 282.84,Z 567.324,A -85,B 0,C 180,E1 -17349.642,E2 -17349.642} C_VEL
LIN {X 0,Y 280.353,Z 575.782,A -85,B 0,C 180,E1 -17351.738,E2 -17351.738} C_VEL
LIN {X 0,Y 278.607,Z 582.72,A -85,B 0,C 180,E1 -17353.89,E2 -17353.89} C_VEL
LIN {X 0,Y 277.186,Z 588.39,A -85,B 0,C 180,E1 -17356.062,E2 -17356.062} C_VEL
LIN {X 0,Y 276.27,Z 592.933,A -85,B 0,C 180,E1 -17358.257,E2 -17358.257} C_VEL
LIN {X 0,Y 275.893,Z 596.436,A -85,B 0,C 180,E1 -17360.469,E2 -17360.469} C_VEL
LIN {X 0,Y 275.989,Z 599.491,A -85,B 0,C 180,E1 -17363.283,E2 -17363.283} C_VEL
LIN {X 0,Y 276.345,Z 600.826,A -85,B 0,C 180,E1 -17365.624,E2 -17365.624} C_VEL
LIN {X 0,Y 276.575,Z 601.082,A -85,B 0,C 180,E1 -17367.087,E2 -17367.087} C_VEL
LIN {X 0,Y 277.089,Z 600.618,A -85,B 0,C 180,E1 -17369.636,E2 -17369.636} C_VEL
LIN {X 0,Y 276.767,Z 601.714,A -85,B 0,C 180,E1 -17371.455,E2 -17371.455} C_VEL
LIN {X 0,Y 276.523,Z 602.037,A -85,B 0,C 180,E1 -17372.913,E2 -17372.913} C_VEL
LIN {X 0,Y 276.274,Z 601.917,A -85,B 0,C 180,E1 -17374.377,E2 -17374.377} C_VEL
LIN {X 0,Y 275.934,Z 600.875,A -85,B 0,C 180,E1 -17376.618,E2 -17376.618} C_VEL
LIN {X 0,Y 275.8,Z 598.933,A -85,B 0,C 180,E1 -17378.794,E2 -17378.794} C_VEL
LIN {X 0,Y 276.217,Z 594.834,A -85,B 0,C 180,E1 -17381.744,E2 -17381.744} C_VEL
LIN {X 0,Y 277.19,Z 590.598,A -85,B 0,C 180,E1 -17383.938,E2 -17383.938} C_VEL
LIN {X 0,Y 278.652,Z 585.302,A -85,B 0,C 180,E1 -17386.107,E2 -17386.107} C_VEL
LIN {X 0,Y 280.465,Z 578.843,A -85,B 0,C 180,E1 -17388.254,E2 -17388.254} C_VEL
LIN {X 0,Y 282.933,Z 571.041,A -85,B 0,C 180,E1 -17390.35,E2 -17390.35} C_VEL
LIN {X 0,Y 286.015,Z 561.576,A -85,B 0,C 180,E1 -17392.387,E2 -17392.387} C_VEL
LIN {X 0,Y 289.271,Z 551.191,A -85,B 0,C 180,E1 -17394.204,E2 -17394.204} C_VEL
LIN {X 0,Y 292.735,Z 539.792,A -85,B 0,C 180,E1 -17395.795,E2 -17395.795} C_VEL
LIN {X 0,Y 296.283,Z 527.235,A -85,B 0,C 180,E1 -17397.169,E2 -17397.169} C_VEL
LIN {X 0,Y 299.178,Z 515.407,A -85,B 0,C 180,E1 -17398.213,E2 -17398.213} C_VEL
LIN {X 0,Y 302.062,Z 501.498,A -85,B 0,C 180,E1 -17399.153,E2 -17399.153} C_VEL
LIN {X 0,Y 304.321,Z 487.566,A -85,B 0,C 180,E1 -17399.865,E2 -17399.865} C_VEL
LIN {X 0,Y 307.882,Z 456.029,A -85,B 0,C 180,E1 -17401.185,E2 -17401.185} C_VEL
LIN {X 0,Y 308.302,Z 443.662,A -85,B 0,C 180,E1 -17401.962,E2 -17401.962} C_VEL
LIN {X 0,Y 308.105,Z 430.663,A -85,B 0,C 180,E1 -17402.999,E2 -17402.999} C_VEL
LIN {X 0,Y 307.513,Z 417.791,A -85,B 0,C 180,E1 -17404.233,E2 -17404.233} C_VEL
LIN {X 0,Y 306.618,Z 406.065,A -85,B 0,C 180,E1 -17405.601,E2 -17405.601} C_VEL
LIN {X 0,Y 305.386,Z 402.334,A -85,B 0,C 180,E1 -17406.434,E2 -17406.434} C_VEL
LIN {X 0,Y 303.097,Z 395.846,A -85,B 0,C 180,E1 -17408.156,E2 -17408.156} C_VEL
LIN {X 0,Y 299.702,Z 386.947,A -85,B 0,C 180,E1 -17411.541,E2 -17411.541} C_VEL
LIN {X 0,Y 298.066,Z 382.591,A -85,B 0,C 180,E1 -17414.386,E2 -17414.386} C_VEL
LIN {X 0,Y 297.77,Z 379.878,A -85,B 0,C 180,E1 -17417.227,E2 -17417.227} C_VEL
LIN {X 0,Y 298.216,Z 379.065,A -85,B 0,C 180,E1 -17418.95,E2 -17418.95} C_VEL
LIN {X 0,Y 299.86,Z 379.557,A -85,B 0,C 180,E1 -17421.727,E2 -17421.727} C_VEL
LIN {X 0,Y 301.399,Z 380.115,A -85,B 0,C 180,E1 -17423.225,E2 -17423.225} C_VEL
LIN {X 0,Y 304.176,Z 382.749,A -85,B 0,C 180,E1 -17425.452,E2 -17425.452} C_VEL
LIN {X 0,Y 307.171,Z 386.161,A -85,B 0,C 180,E1 -17427.322,E2 -17427.322} C_VEL
LIN {X 0,Y 309.114,Z 388.459,A -85,B 0,C 180,E1 -17428.354,E2 -17428.354} C_VEL
LIN {X 0,Y 312.502,Z 395.063,A -85,B 0,C 180,E1 -17430.138,E2 -17430.138} C_VEL
LIN {X 0,Y 313.569,Z 397.355,A -85,B 0,C 180,E1 -17430.652,E2 -17430.652} C_VEL
LIN {X 0,Y 308.811,Z 434.566,A -85,B 0,C 180,E1 -17432.237,E2 -17432.237} C_VEL
LIN {X 0,Y 307.12,Z 451.441,A -85,B 0,C 180,E1 -17433.117,E2 -17433.117} C_VEL
LIN {X 0,Y 305.356,Z 464.545,A -85,B 0,C 180,E1 -17434.068,E2 -17434.068} C_VEL
LIN {X 0,Y 302.95,Z 477.799,A -85,B 0,C 180,E1 -17435.318,E2 -17435.318} C_VEL
LIN {X 0,Y 299.999,Z 490.646,A -85,B 0,C 180,E1 -17436.896,E2 -17436.896} C_VEL
LIN {X 0,Y 297.12,Z 500.915,A -85,B 0,C 180,E1 -17438.491,E2 -17438.491} C_VEL
LIN {X 0,Y 294.437,Z 509.366,A -85,B 0,C 180,E1 -17440.114,E2 -17440.114} C_VEL
LIN {X 0,Y 291.481,Z 517.687,A -85,B 0,C 180,E1 -17442.096,E2 -17442.096} C_VEL
LIN {X 0,Y 288.333,Z 525.358,A -85,B 0,C 180,E1 -17444.447,E2 -17444.447} C_VEL
LIN {X 0,Y 285.947,Z 530.491,A -85,B 0,C 180,E1 -17446.497,E2 -17446.497} C_VEL
LIN {X 0,Y 283.811,Z 534.462,A -85,B 0,C 180,E1 -17448.573,E2 -17448.573} C_VEL
LIN {X 0,Y 282.597,Z 536.472,A -85,B 0,C 180,E1 -17449.974,E2 -17449.974} C_VEL
LIN {X 0,Y 281.433,Z 538.073,A -85,B 0,C 180,E1 -17451.382,E2 -17451.382} C_VEL
LIN {X 0,Y 280.461,Z 539.236,A -85,B 0,C 180,E1 -17452.802,E2 -17452.802} C_VEL
LIN {X 0,Y 279.634,Z 539.94,A -85,B 0,C 180,E1 -17454.23,E2 -17454.23} C_VEL
LIN {X 0,Y 278.868,Z 540.236,A -85,B 0,C 180,E1 -17455.663,E2 -17455.663} C_VEL
LIN {X 0,Y 278.308,Z 540.113,A -85,B 0,C 180,E1 -17457.104,E2 -17457.104} C_VEL
LIN {X 0,Y 277.798,Z 539.58,A -85,B 0,C 180,E1 -17458.55,E2 -17458.55} C_VEL
LIN {X 0,Y 277.49,Z 538.579,A -85,B 0,C 180,E1 -17459.999,E2 -17459.999} C_VEL
LIN {X 0,Y 276.969,Z 537.198,A -85,B 0,C 180,E1 -17461.453,E2 -17461.453} C_VEL
LIN {X 0,Y 276.725,Z 534.259,A -85,B 0,C 180,E1 -17463.64,E2 -17463.64} C_VEL
LIN {X 0,Y 276.886,Z 530.261,A -85,B 0,C 180,E1 -17465.827,E2 -17465.827} C_VEL
LIN {X 0,Y 277.02,Z 524.271,A -85,B 0,C 180,E1 -17468.337,E2 -17468.337} C_VEL
LIN {X 0,Y 277.402,Z 517.395,A -85,B 0,C 180,E1 -17470.583,E2 -17470.583} C_VEL
LIN {X 0,Y 277.934,Z 509.079,A -85,B 0,C 180,E1 -17472.782,E2 -17472.782} C_VEL
LIN {X 0,Y 278.573,Z 500.618,A -85,B 0,C 180,E1 -17474.612,E2 -17474.612} C_VEL
LIN {X 0,Y 279.414,Z 489.151,A -85,B 0,C 180,E1 -17476.633,E2 -17476.633} C_VEL
LIN {X 0,Y 280.155,Z 477.539,A -85,B 0,C 180,E1 -17478.274,E2 -17478.274} C_VEL
LIN {X 0,Y 281.023,Z 464.572,A -85,B 0,C 180,E1 -17479.731,E2 -17479.731} C_VEL
LIN {X 0,Y 281.74,Z 450.709,A -85,B 0,C 180,E1 -17480.917,E2 -17480.917} C_VEL
LIN {X 0,Y 282.251,Z 436.831,A -85,B 0,C 180,E1 -17481.787,E2 -17481.787} C_VEL
LIN {X 0,Y 282.634,Z 414.895,A -85,B 0,C 180,E1 -17482.684,E2 -17482.684} C_VEL
LIN {X 0,Y 284.172,Z 369.532,A -85,B 0,C 180,E1 -17484.376,E2 -17484.376} C_VEL
LIN {X 0,Y 277.377,Z 346.932,A -85,B 0,C 180,E1 -17485.564,E2 -17485.564} C_VEL
LIN {X 0,Y 277.29,Z 346.946,A -85,B 0,C 180,E1 -17488.786,E2 -17488.786} C_VEL
LIN {X 0,Y 277.253,Z 346.948,A -85,B 0,C 180,E1 -17493.227,E2 -17493.227} C_VEL
LIN {X 0,Y 277.278,Z 346.943,A -85,B 0,C 180,E1 -17495.798,E2 -17495.798} C_VEL
LIN {X 0,Y 277.231,Z 346.949,A -85,B 0,C 180,E1 -17499.328,E2 -17499.328} C_VEL
LIN {X 0,Y 277.215,Z 346.953,A -85,B 0,C 180,E1 -17503.196,E2 -17503.196} C_VEL
LIN {X 0,Y 277.216,Z 346.951,A -85,B 0,C 180,E1 -17507.324,E2 -17507.324} C_VEL
LIN {X 0,Y 277.273,Z 346.944,A -85,B 0,C 180,E1 -17511.789,E2 -17511.789} C_VEL
LIN {X 0,Y 277.301,Z 346.942,A -85,B 0,C 180,E1 -17514.344,E2 -17514.344} C_VEL
LIN {X 0,Y 277.241,Z 346.948,A -85,B 0,C 180,E1 -17517.836,E2 -17517.836} C_VEL
LIN {X 0,Y 277.265,Z 346.946,A -85,B 0,C 180,E1 -17521.21,E2 -17521.21} C_VEL
LIN {X 0,Y 277.309,Z 346.942,A -85,B 0,C 180,E1 -17524.479,E2 -17524.479} C_VEL
LIN {X 0,Y 277.283,Z 346.943,A -85,B 0,C 180,E1 -17527.655,E2 -17527.655} C_VEL
LIN {X 0,Y 277.342,Z 346.938,A -85,B 0,C 180,E1 -17530.766,E2 -17530.766} C_VEL
LIN {X 0,Y 277.432,Z 346.924,A -85,B 0,C 180,E1 -17535.326,E2 -17535.326} C_VEL
LIN {X 0,Y 277.504,Z 346.915,A -85,B 0,C 180,E1 -17539.789,E2 -17539.789} C_VEL
LIN {X 0,Y 277.651,Z 346.899,A -85,B 0,C 180,E1 -17542.729,E2 -17542.729} C_VEL
LIN {X 0,Y 277.819,Z 346.878,A -85,B 0,C 180,E1 -17548.551,E2 -17548.551} C_VEL
LIN {X 0,Y 277.819,Z 346.875,A -85,B 0,C 180,E1 -17551.45,E2 -17551.45} C_VEL
LIN {X 0,Y 277.651,Z 346.896,A -85,B 0,C 180,E1 -17557.271,E2 -17557.271} C_VEL
LIN {X 0,Y 277.504,Z 346.918,A -85,B 0,C 180,E1 -17560.212,E2 -17560.212} C_VEL
LIN {X 0,Y 277.432,Z 346.925,A -85,B 0,C 180,E1 -17564.675,E2 -17564.675} C_VEL
LIN {X 0,Y 277.343,Z 346.935,A -85,B 0,C 180,E1 -17569.234,E2 -17569.234} C_VEL
LIN {X 0,Y 277.317,Z 346.943,A -85,B 0,C 180,E1 -17574.171,E2 -17574.171} C_VEL
LIN {X 0,Y 277.323,Z 346.938,A -85,B 0,C 180,E1 -17577.505,E2 -17577.505} C_VEL
LIN {X 0,Y 277.27,Z 346.947,A -85,B 0,C 180,E1 -17580.482,E2 -17580.482} C_VEL
LIN {X 0,Y 277.253,Z 346.948,A -85,B 0,C 180,E1 -17583.895,E2 -17583.895} C_VEL
LIN {X 0,Y 277.28,Z 346.944,A -85,B 0,C 180,E1 -17587.468,E2 -17587.468} C_VEL
LIN {X 0,Y 277.209,Z 346.951,A -85,B 0,C 180,E1 -17591.237,E2 -17591.237} C_VEL
LIN {X 0,Y 277.201,Z 346.953,A -85,B 0,C 180,E1 -17595.227,E2 -17595.227} C_VEL
LIN {X 0,Y 277.222,Z 346.951,A -85,B 0,C 180,E1 -17599.513,E2 -17599.513} C_VEL
LIN {X 0,Y 277.274,Z 346.944,A -85,B 0,C 180,E1 -17602.533,E2 -17602.533} C_VEL
LIN {X 0,Y 277.248,Z 346.951,A -85,B 0,C 180,E1 -17606.105,E2 -17606.105} C_VEL
LIN {X 0,Y 277.295,Z 346.945,A -85,B 0,C 180,E1 -17608.088,E2 -17608.088} C_VEL
LIN {X 0,Y 284.778,Z 370.712,A -85,B 0,C 180,E1 -17609.359,E2 -17609.359} C_VEL
LIN {X 0,Y 282.874,Z 432.18,A -85,B 0,C 180,E1 -17611.555,E2 -17611.555} C_VEL
LIN {X 0,Y 282.508,Z 445.878,A -85,B 0,C 180,E1 -17612.298,E2 -17612.298} C_VEL
LIN {X 0,Y 281.809,Z 459.31,A -85,B 0,C 180,E1 -17613.328,E2 -17613.328} C_VEL
LIN {X 0,Y 281.064,Z 471.946,A -85,B 0,C 180,E1 -17614.601,E2 -17614.601} C_VEL
LIN {X 0,Y 280.18,Z 483.964,A -85,B 0,C 180,E1 -17616.142,E2 -17616.142} C_VEL
LIN {X 0,Y 279.291,Z 494.531,A -85,B 0,C 180,E1 -17617.825,E2 -17617.825} C_VEL
LIN {X 0,Y 278.557,Z 504.147,A -85,B 0,C 180,E1 -17619.702,E2 -17619.702} C_VEL
LIN {X 0,Y 277.909,Z 512.041,A -85,B 0,C 180,E1 -17621.573,E2 -17621.573} C_VEL
LIN {X 0,Y 277.374,Z 519.728,A -85,B 0,C 180,E1 -17623.817,E2 -17623.817} C_VEL
LIN {X 0,Y 277.007,Z 525.857,A -85,B 0,C 180,E1 -17626.054,E2 -17626.054} C_VEL
LIN {X 0,Y 276.834,Z 530.68,A -85,B 0,C 180,E1 -17628.283,E2 -17628.283} C_VEL
LIN {X 0,Y 276.915,Z 534.58,A -85,B 0,C 180,E1 -17630.704,E2 -17630.704} C_VEL
LIN {X 0,Y 276.36,Z 536.099,A -85,B 0,C 180,E1 -17631.883,E2 -17631.883} C_VEL
LIN {X 0,Y 273.782,Z 538.28,A -85,B 0,C 180,E1 -17633.828,E2 -17633.828} C_VEL
LIN {X 0,Y 271.389,Z 539.697,A -85,B 0,C 180,E1 -17635.831,E2 -17635.831} C_VEL
LIN {X 0,Y 271.137,Z 539.984,A -85,B 0,C 180,E1 -17637.077,E2 -17637.077} C_VEL
LIN {X 0,Y 271.762,Z 540.005,A -85,B 0,C 180,E1 -17638.519,E2 -17638.519} C_VEL
LIN {X 0,Y 272.476,Z 539.613,A -85,B 0,C 180,E1 -17640.001,E2 -17640.001} C_VEL
LIN {X 0,Y 274.324,Z 537.489,A -85,B 0,C 180,E1 -17642.938,E2 -17642.938} C_VEL
LIN {X 0,Y 276.038,Z 534.76,A -85,B 0,C 180,E1 -17645.113,E2 -17645.113} C_VEL
LIN {X 0,Y 278.008,Z 530.965,A -85,B 0,C 180,E1 -17647.262,E2 -17647.262} C_VEL
LIN {X 0,Y 280.302,Z 525.99,A -85,B 0,C 180,E1 -17649.38,E2 -17649.38} C_VEL
LIN {X 0,Y 282.951,Z 519.699,A -85,B 0,C 180,E1 -17651.462,E2 -17651.462} C_VEL
LIN {X 0,Y 285.724,Z 511.919,A -85,B 0,C 180,E1 -17653.514,E2 -17653.514} C_VEL
LIN {X 0,Y 288.31,Z 503.928,A -85,B 0,C 180,E1 -17655.192,E2 -17655.192} C_VEL
LIN {X 0,Y 291.302,Z 493.259,A -85,B 0,C 180,E1 -17657.01,E2 -17657.01} C_VEL
LIN {X 0,Y 293.898,Z 482.426,A -85,B 0,C 180,E1 -17658.473,E2 -17658.473} C_VEL
LIN {X 0,Y 296.261,Z 470.218,A -85,B 0,C 180,E1 -17659.758,E2 -17659.758} C_VEL
LIN {X 0,Y 298.226,Z 456.564,A -85,B 0,C 180,E1 -17660.882,E2 -17660.882} C_VEL
LIN {X 0,Y 299.539,Z 444.003,A -85,B 0,C 180,E1 -17661.643,E2 -17661.643} C_VEL
LIN {X 0,Y 302.212,Z 415.833,A -85,B 0,C 180,E1 -17662.853,E2 -17662.853} C_VEL
LIN {X 0,Y 304.411,Z 396.33,A -85,B 0,C 180,E1 -17663.635,E2 -17663.635} C_VEL
LIN {X 0,Y 300.093,Z 388.039,A -85,B 0,C 180,E1 -17665.54,E2 -17665.54} C_VEL
LIN {X 0,Y 296.888,Z 382.69,A -85,B 0,C 180,E1 -17667.107,E2 -17667.107} C_VEL
LIN {X 0,Y 294.868,Z 379.391,A -85,B 0,C 180,E1 -17668.235,E2 -17668.235} C_VEL
LIN {X 0,Y 292.68,Z 375.765,A -85,B 0,C 180,E1 -17669.628,E2 -17669.628} C_VEL
LIN {X 0,Y 290.276,Z 372.763,A -85,B 0,C 180,E1 -17671.303,E2 -17671.303} C_VEL
LIN {X 0,Y 289.242,Z 370.81,A -85,B 0,C 180,E1 -17672.235,E2 -17672.235} C_VEL
LIN {X 0,Y 286.837,Z 368.223,A -85,B 0,C 180,E1 -17674.718,E2 -17674.718} C_VEL
LIN {X 0,Y 286.31,Z 367.231,A -85,B 0,C 180,E1 -17675.587,E2 -17675.587} C_VEL
LIN {X 0,Y 285.156,Z 366.093,A -85,B 0,C 180,E1 -17678.037,E2 -17678.037} C_VEL
LIN {X 0,Y 284.821,Z 366.399,A -85,B 0,C 180,E1 -17680.371,E2 -17680.371} C_VEL
LIN {X 0,Y 285.827,Z 368.722,A -85,B 0,C 180,E1 -17683.982,E2 -17683.982} C_VEL
LIN {X 0,Y 287.268,Z 370.472,A -85,B 0,C 180,E1 -17685.909,E2 -17685.909} C_VEL
LIN {X 0,Y 290.663,Z 375.832,A -85,B 0,C 180,E1 -17689.061,E2 -17689.061} C_VEL
LIN {X 0,Y 293.838,Z 380.779,A -85,B 0,C 180,E1 -17691.209,E2 -17691.209} C_VEL
LIN {X 0,Y 294.483,Z 382.361,A -85,B 0,C 180,E1 -17691.646,E2 -17691.646} C_VEL
LIN {X 0,Y 297.422,Z 394.046,A -85,B 0,C 180,E1 -17693.831,E2 -17693.831} C_VEL
LIN {X 0,Y 297.984,Z 397.201,A -85,B 0,C 180,E1 -17694.281,E2 -17694.281} C_VEL
LIN {X 0,Y 298.584,Z 411.861,A -85,B 0,C 180,E1 -17695.637,E2 -17695.637} C_VEL
LIN {X 0,Y 299.077,Z 433.288,A -85,B 0,C 180,E1 -17697.334,E2 -17697.334} C_VEL
LIN {X 0,Y 299.046,Z 449.637,A -85,B 0,C 180,E1 -17698.413,E2 -17698.413} C_VEL
LIN {X 0,Y 298.69,Z 459.98,A -85,B 0,C 180,E1 -17699.001,E2 -17699.001} C_VEL
LIN {X 0,Y 295.161,Z 493.055,A -85,B 0,C 180,E1 -17700.342,E2 -17700.342} C_VEL
LIN {X 0,Y 292.869,Z 506.871,A -85,B 0,C 180,E1 -17701.122,E2 -17701.122} C_VEL
LIN {X 0,Y 289.866,Z 520.747,A -85,B 0,C 180,E1 -17702.177,E2 -17702.177} C_VEL
LIN {X 0,Y 286.682,Z 533.295,A -85,B 0,C 180,E1 -17703.423,E2 -17703.423} C_VEL
LIN {X 0,Y 283.371,Z 544.778,A -85,B 0,C 180,E1 -17704.866,E2 -17704.866} C_VEL
LIN {X 0,Y 280.502,Z 554.278,A -85,B 0,C 180,E1 -17706.366,E2 -17706.366} C_VEL
LIN {X 0,Y 277.221,Z 564.806,A -85,B 0,C 180,E1 -17708.432,E2 -17708.432} C_VEL
LIN {X 0,Y 274.411,Z 573.487,A -85,B 0,C 180,E1 -17710.552,E2 -17710.552} C_VEL
LIN {X 0,Y 272.12,Z 580.992,A -85,B 0,C 180,E1 -17712.863,E2 -17712.863} C_VEL
LIN {X 0,Y 270.647,Z 586.469,A -85,B 0,C 180,E1 -17714.949,E2 -17714.949} C_VEL
LIN {X 0,Y 269.562,Z 591.171,A -85,B 0,C 180,E1 -17717.196,E2 -17717.196} C_VEL
LIN {X 0,Y 268.92,Z 594.843,A -85,B 0,C 180,E1 -17719.459,E2 -17719.459} C_VEL
LIN {X 0,Y 268.803,Z 598.198,A -85,B 0,C 180,E1 -17722.488,E2 -17722.488} C_VEL
LIN {X 0,Y 269.008,Z 599.273,A -85,B 0,C 180,E1 -17724.001,E2 -17724.001} C_VEL
LIN {X 0,Y 269.278,Z 599.891,A -85,B 0,C 180,E1 -17725.509,E2 -17725.509} C_VEL
LIN {X 0,Y 269.526,Z 600.038,A -85,B 0,C 180,E1 -17727.01,E2 -17727.01} C_VEL
LIN {X 0,Y 270.112,Z 599.301,A -85,B 0,C 180,E1 -17729.627,E2 -17729.627} C_VEL
LIN {X 0,Y 269.781,Z 600.494,A -85,B 0,C 180,E1 -17731.493,E2 -17731.493} C_VEL
LIN {X 0,Y 269.482,Z 600.938,A -85,B 0,C 180,E1 -17732.99,E2 -17732.99} C_VEL
LIN {X 0,Y 269.21,Z 600.9,A -85,B 0,C 180,E1 -17734.492,E2 -17734.492} C_VEL
LIN {X 0,Y 268.867,Z 600.123,A -85,B 0,C 180,E1 -17736.634,E2 -17736.634} C_VEL
LIN {X 0,Y 268.716,Z 598.234,A -85,B 0,C 180,E1 -17739.028,E2 -17739.028} C_VEL
LIN {X 0,Y 269.016,Z 595.48,A -85,B 0,C 180,E1 -17741.299,E2 -17741.299} C_VEL
LIN {X 0,Y 269.878,Z 591.784,A -85,B 0,C 180,E1 -17743.554,E2 -17743.554} C_VEL
LIN {X 0,Y 271.222,Z 587.083,A -85,B 0,C 180,E1 -17745.788,E2 -17745.788} C_VEL
LIN {X 0,Y 272.974,Z 581.276,A -85,B 0,C 180,E1 -17747.996,E2 -17747.996} C_VEL
LIN {X 0,Y 275.376,Z 574.252,A -85,B 0,C 180,E1 -17750.154,E2 -17750.154} C_VEL
LIN {X 0,Y 278.379,Z 565.817,A -85,B 0,C 180,E1 -17752.253,E2 -17752.253} C_VEL
LIN {X 0,Y 281.933,Z 555.59,A -85,B 0,C 180,E1 -17754.287,E2 -17754.287} C_VEL
LIN {X 0,Y 285.702,Z 544.297,A -85,B 0,C 180,E1 -17756.085,E2 -17756.085} C_VEL
LIN {X 0,Y 289.684,Z 531.671,A -85,B 0,C 180,E1 -17757.645,E2 -17757.645} C_VEL
LIN {X 0,Y 293.148,Z 519.422,A -85,B 0,C 180,E1 -17758.848,E2 -17758.848} C_VEL
LIN {X 0,Y 296.321,Z 506.049,A -85,B 0,C 180,E1 -17759.872,E2 -17759.872} C_VEL
LIN {X 0,Y 299.217,Z 491.248,A -85,B 0,C 180,E1 -17760.721,E2 -17760.721} C_VEL
LIN {X 0,Y 303.432,Z 458.399,A -85,B 0,C 180,E1 -17762.138,E2 -17762.138} C_VEL
LIN {X 0,Y 304.062,Z 445.549,A -85,B 0,C 180,E1 -17762.966,E2 -17762.966} C_VEL
LIN {X 0,Y 304.058,Z 432.679,A -85,B 0,C 180,E1 -17764.035,E2 -17764.035} C_VEL
LIN {X 0,Y 303.717,Z 420.236,A -85,B 0,C 180,E1 -17765.274,E2 -17765.274} C_VEL
LIN {X 0,Y 303.177,Z 410.434,A -85,B 0,C 180,E1 -17766.457,E2 -17766.457} C_VEL
LIN {X 0,Y 301.993,Z 406.738,A -85,B 0,C 180,E1 -17767.357,E2 -17767.357} C_VEL
LIN {X 0,Y 300.46,Z 401.802,A -85,B 0,C 180,E1 -17768.701,E2 -17768.701} C_VEL
LIN {X 0,Y 297.499,Z 393.198,A -85,B 0,C 180,E1 -17772.049,E2 -17772.049} C_VEL
LIN {X 0,Y 296.158,Z 388.962,A -85,B 0,C 180,E1 -17774.917,E2 -17774.917} C_VEL
LIN {X 0,Y 296.142,Z 386.467,A -85,B 0,C 180,E1 -17777.771,E2 -17777.771} C_VEL
LIN {X 0,Y 296.632,Z 385.985,A -85,B 0,C 180,E1 -17779.303,E2 -17779.303} C_VEL
LIN {X 0,Y 298.892,Z 386.598,A -85,B 0,C 180,E1 -17782.517,E2 -17782.517} C_VEL
LIN {X 0,Y 299.782,Z 387.303,A -85,B 0,C 180,E1 -17783.397,E2 -17783.397} C_VEL
LIN {X 0,Y 301.994,Z 389.33,A -85,B 0,C 180,E1 -17785.182,E2 -17785.182} C_VEL
LIN {X 0,Y 304.828,Z 392.699,A -85,B 0,C 180,E1 -17787.048,E2 -17787.048} C_VEL
LIN {X 0,Y 306.36,Z 394.64,A -85,B 0,C 180,E1 -17787.916,E2 -17787.916} C_VEL
LIN {X 0,Y 309.303,Z 400.659,A -85,B 0,C 180,E1 -17789.594,E2 -17789.594} C_VEL
LIN {X 0,Y 309.433,Z 401.148,A -85,B 0,C 180,E1 -17789.68,E2 -17789.68} C_VEL
LIN {X 0,Y 304.668,Z 435.843,A -85,B 0,C 180,E1 -17791.187,E2 -17791.187} C_VEL
LIN {X 0,Y 302.723,Z 453.292,A -85,B 0,C 180,E1 -17792.126,E2 -17792.126} C_VEL
LIN {X 0,Y 300.85,Z 465.942,A -85,B 0,C 180,E1 -17793.07,E2 -17793.07} C_VEL
LIN {X 0,Y 298.515,Z 477.86,A -85,B 0,C 180,E1 -17794.2,E2 -17794.2} C_VEL
LIN {X 0,Y 296.04,Z 488.345,A -85,B 0,C 180,E1 -17795.452,E2 -17795.452} C_VEL
LIN {X 0,Y 293.496,Z 497.246,A -85,B 0,C 180,E1 -17796.727,E2 -17796.727} C_VEL
LIN {X 0,Y 290.559,Z 506.465,A -85,B 0,C 180,E1 -17798.354,E2 -17798.354} C_VEL
LIN {X 0,Y 287.217,Z 515.554,A -85,B 0,C 180,E1 -17800.338,E2 -17800.338} C_VEL
LIN {X 0,Y 283.717,Z 523.905,A -85,B 0,C 180,E1 -17802.707,E2 -17802.707} C_VEL
LIN {X 0,Y 281.009,Z 529.563,A -85,B 0,C 180,E1 -17804.775,E2 -17804.775} C_VEL
LIN {X 0,Y 278.579,Z 533.997,A -85,B 0,C 180,E1 -17806.876,E2 -17806.876} C_VEL
LIN {X 0,Y 277.099,Z 536.317,A -85,B 0,C 180,E1 -17808.293,E2 -17808.293} C_VEL
LIN {X 0,Y 275.81,Z 538.195,A -85,B 0,C 180,E1 -17809.725,E2 -17809.725} C_VEL
LIN {X 0,Y 274.603,Z 539.647,A -85,B 0,C 180,E1 -17811.166,E2 -17811.166} C_VEL
LIN {X 0,Y 272.693,Z 541.185,A -85,B 0,C 180,E1 -17814.082,E2 -17814.082} C_VEL
LIN {X 0,Y 271.886,Z 541.36,A -85,B 0,C 180,E1 -17815.552,E2 -17815.552} C_VEL
LIN {X 0,Y 271.301,Z 541.078,A -85,B 0,C 180,E1 -17817.029,E2 -17817.029} C_VEL
LIN {X 0,Y 270.773,Z 540.373,A -85,B 0,C 180,E1 -17818.512,E2 -17818.512} C_VEL
LIN {X 0,Y 270.408,Z 539.26,A -85,B 0,C 180,E1 -17819.999,E2 -17819.999} C_VEL
LIN {X 0,Y 269.739,Z 536.792,A -85,B 0,C 180,E1 -17822.239,E2 -17822.239} C_VEL
LIN {X 0,Y 269.711,Z 533.279,A -85,B 0,C 180,E1 -17824.483,E2 -17824.483} C_VEL
LIN {X 0,Y 269.874,Z 528.677,A -85,B 0,C 180,E1 -17826.729,E2 -17826.729} C_VEL
LIN {X 0,Y 270.034,Z 522.839,A -85,B 0,C 180,E1 -17828.983,E2 -17828.983} C_VEL
LIN {X 0,Y 270.461,Z 515.537,A -85,B 0,C 180,E1 -17831.238,E2 -17831.238} C_VEL
LIN {X 0,Y 271.018,Z 506.531,A -85,B 0,C 180,E1 -17833.496,E2 -17833.496} C_VEL
LIN {X 0,Y 271.84,Z 496.327,A -85,B 0,C 180,E1 -17835.558,E2 -17835.558} C_VEL
LIN {X 0,Y 272.465,Z 486.374,A -85,B 0,C 180,E1 -17837.209,E2 -17837.209} C_VEL
LIN {X 0,Y 273.296,Z 475.053,A -85,B 0,C 180,E1 -17838.75,E2 -17838.75} C_VEL
LIN {X 0,Y 274.079,Z 463.005,A -85,B 0,C 180,E1 -17840.057,E2 -17840.057} C_VEL
LIN {X 0,Y 274.751,Z 449.775,A -85,B 0,C 180,E1 -17841.18,E2 -17841.18} C_VEL
LIN {X 0,Y 275.254,Z 436.025,A -85,B 0,C 180,E1 -17842.024,E2 -17842.024} C_VEL
LIN {X 0,Y 275.994,Z 402.052,A -85,B 0,C 180,E1 -17843.398,E2 -17843.398} C_VEL
LIN {X 0,Y 277.195,Z 370.929,A -85,B 0,C 180,E1 -17844.598,E2 -17844.598} C_VEL
LIN {X 0,Y 270.334,Z 347.809,A -85,B 0,C 180,E1 -17845.876,E2 -17845.876} C_VEL
LIN {X 0,Y 270.229,Z 347.82,A -85,B 0,C 180,E1 -17849.612,E2 -17849.612} C_VEL
LIN {X 0,Y 270.215,Z 347.823,A -85,B 0,C 180,E1 -17853.666,E2 -17853.666} C_VEL
LIN {X 0,Y 270.214,Z 347.827,A -85,B 0,C 180,E1 -17856.741,E2 -17856.741} C_VEL
LIN {X 0,Y 270.167,Z 347.832,A -85,B 0,C 180,E1 -17861.028,E2 -17861.028} C_VEL
LIN {X 0,Y 270.164,Z 347.829,A -85,B 0,C 180,E1 -17865.382,E2 -17865.382} C_VEL
LIN {X 0,Y 270.172,Z 347.829,A -85,B 0,C 180,E1 -17869.434,E2 -17869.434} C_VEL
LIN {X 0,Y 270.253,Z 347.818,A -85,B 0,C 180,E1 -17873.722,E2 -17873.722} C_VEL
LIN {X 0,Y 270.201,Z 347.827,A -85,B 0,C 180,E1 -17876.892,E2 -17876.892} C_VEL
LIN {X 0,Y 270.192,Z 347.829,A -85,B 0,C 180,E1 -17880.382,E2 -17880.382} C_VEL
LIN {X 0,Y 270.259,Z 347.816,A -85,B 0,C 180,E1 -17883.763,E2 -17883.763} C_VEL
LIN {X 0,Y 270.23,Z 347.823,A -85,B 0,C 180,E1 -17887.039,E2 -17887.039} C_VEL
LIN {X 0,Y 270.299,Z 347.815,A -85,B 0,C 180,E1 -17890.244,E2 -17890.244} C_VEL
LIN {X 0,Y 270.4,Z 347.802,A -85,B 0,C 180,E1 -17894.935,E2 -17894.935} C_VEL
LIN {X 0,Y 270.439,Z 347.795,A -85,B 0,C 180,E1 -17899.519,E2 -17899.519} C_VEL
LIN {X 0,Y 270.609,Z 347.778,A -85,B 0,C 180,E1 -17902.539,E2 -17902.539} C_VEL
LIN {X 0,Y 270.785,Z 347.755,A -85,B 0,C 180,E1 -17908.513,E2 -17908.513} C_VEL
LIN {X 0,Y 270.785,Z 347.751,A -85,B 0,C 180,E1 -17911.487,E2 -17911.487} C_VEL
LIN {X 0,Y 270.609,Z 347.773,A -85,B 0,C 180,E1 -17917.462,E2 -17917.462} C_VEL
LIN {X 0,Y 270.439,Z 347.799,A -85,B 0,C 180,E1 -17920.481,E2 -17920.481} C_VEL
LIN {X 0,Y 270.401,Z 347.8,A -85,B 0,C 180,E1 -17925.065,E2 -17925.065} C_VEL
LIN {X 0,Y 270.3,Z 347.814,A -85,B 0,C 180,E1 -17929.756,E2 -17929.756} C_VEL
LIN {X 0,Y 270.272,Z 347.816,A -85,B 0,C 180,E1 -17934.586,E2 -17934.586} C_VEL
LIN {X 0,Y 270.268,Z 347.819,A -85,B 0,C 180,E1 -17937.909,E2 -17937.909} C_VEL
LIN {X 0,Y 270.183,Z 347.827,A -85,B 0,C 180,E1 -17941.349,E2 -17941.349} C_VEL
LIN {X 0,Y 270.214,Z 347.823,A -85,B 0,C 180,E1 -17944.904,E2 -17944.904} C_VEL
LIN {X 0,Y 270.221,Z 347.823,A -85,B 0,C 180,E1 -17948.718,E2 -17948.718} C_VEL
LIN {X 0,Y 270.165,Z 347.828,A -85,B 0,C 180,E1 -17953.25,E2 -17953.25} C_VEL
LIN {X 0,Y 270.172,Z 347.83,A -85,B 0,C 180,E1 -17957.443,E2 -17957.443} C_VEL
LIN {X 0,Y 270.207,Z 347.823,A -85,B 0,C 180,E1 -17961.375,E2 -17961.375} C_VEL
LIN {X 0,Y 270.204,Z 347.825,A -85,B 0,C 180,E1 -17965.096,E2 -17965.096} C_VEL
LIN {X 0,Y 270.255,Z 347.821,A -85,B 0,C 180,E1 -17967.759,E2 -17967.759} C_VEL
LIN {X 0,Y 277.847,Z 372.123,A -85,B 0,C 180,E1 -17969.098,E2 -17969.098} C_VEL
LIN {X 0,Y 275.888,Z 432.408,A -85,B 0,C 180,E1 -17971.314,E2 -17971.314} C_VEL
LIN {X 0,Y 275.513,Z 445.877,A -85,B 0,C 180,E1 -17972.049,E2 -17972.049} C_VEL
LIN {X 0,Y 274.819,Z 459.603,A -85,B 0,C 180,E1 -17973.114,E2 -17973.114} C_VEL
LIN {X 0,Y 274.074,Z 471.84,A -85,B 0,C 180,E1 -17974.361,E2 -17974.361} C_VEL
LIN {X 0,Y 273.167,Z 483.664,A -85,B 0,C 180,E1 -17975.895,E2 -17975.895} C_VEL
LIN {X 0,Y 272.269,Z 494.522,A -85,B 0,C 180,E1 -17977.632,E2 -17977.632} C_VEL
LIN {X 0,Y 271.498,Z 504.204,A -85,B 0,C 180,E1 -17979.546,E2 -17979.546} C_VEL
LIN {X 0,Y 270.72,Z 513.702,A -85,B 0,C 180,E1 -17981.85,E2 -17981.85} C_VEL
LIN {X 0,Y 270.169,Z 522.125,A -85,B 0,C 180,E1 -17984.448,E2 -17984.448} C_VEL
LIN {X 0,Y 269.873,Z 527.301,A -85,B 0,C 180,E1 -17986.446,E2 -17986.446} C_VEL
LIN {X 0,Y 269.741,Z 532.035,A -85,B 0,C 180,E1 -17988.732,E2 -17988.732} C_VEL
LIN {X 0,Y 269.878,Z 535.578,A -85,B 0,C 180,E1 -17991.012,E2 -17991.012} C_VEL
LIN {X 0,Y 270.06,Z 537.32,A -85,B 0,C 180,E1 -17992.524,E2 -17992.524} C_VEL
LIN {X 0,Y 270.279,Z 538.651,A -85,B 0,C 180,E1 -17994.031,E2 -17994.031} C_VEL
LIN {X 0,Y 270.593,Z 539.557,A -85,B 0,C 180,E1 -17995.532,E2 -17995.532} C_VEL
LIN {X 0,Y 271.137,Z 539.984,A -85,B 0,C 180,E1 -17997.077,E2 -17997.077} C_VEL
LIN {X 0,Y 270.997,Z 540.141,A -85,B 0,C 180,E1 -17998.326,E2 -17998.326} C_VEL
LIN {X 0,Y 269.216,Z 540.083,A -85,B 0,C 180,E1 -18000.397,E2 -18000.397} C_VEL
LIN {X 0,Y 267.838,Z 539.623,A -85,B 0,C 180,E1 -18002.064,E2 -18002.064} C_VEL
LIN {X 0,Y 267.666,Z 538.83,A -85,B 0,C 180,E1 -18003.316,E2 -18003.316} C_VEL
LIN {X 0,Y 267.882,Z 538.411,A -85,B 0,C 180,E1 -18003.727,E2 -18003.727} C_VEL
LIN {X 0,Y 269.831,Z 535.622,A -85,B 0,C 180,E1 -18005.981,E2 -18005.981} C_VEL
LIN {X 0,Y 271.964,Z 531.814,A -85,B 0,C 180,E1 -18008.172,E2 -18008.172} C_VEL
LIN {X 0,Y 274.463,Z 526.807,A -85,B 0,C 180,E1 -18010.326,E2 -18010.326} C_VEL
LIN {X 0,Y 277.742,Z 519.24,A -85,B 0,C 180,E1 -18012.793,E2 -18012.793} C_VEL
LIN {X 0,Y 280.841,Z 511.127,A -85,B 0,C 180,E1 -18014.863,E2 -18014.863} C_VEL
LIN {X 0,Y 284.266,Z 500.965,A -85,B 0,C 180,E1 -18016.888,E2 -18016.888} C_VEL
LIN {X 0,Y 287.2,Z 490.385,A -85,B 0,C 180,E1 -18018.55,E2 -18018.55} C_VEL
LIN {X 0,Y 289.683,Z 480.144,A -85,B 0,C 180,E1 -18019.856,E2 -18019.856} C_VEL
LIN {X 0,Y 292.226,Z 467.17,A -85,B 0,C 180,E1 -18021.147,E2 -18021.147} C_VEL
LIN {X 0,Y 294.023,Z 454.558,A -85,B 0,C 180,E1 -18022.116,E2 -18022.116} C_VEL
LIN {X 0,Y 295.314,Z 441.305,A -85,B 0,C 180,E1 -18022.862,E2 -18022.862} C_VEL
LIN {X 0,Y 299.221,Z 406.583,A -85,B 0,C 180,E1 -18024.339,E2 -18024.339} C_VEL
LIN {X 0,Y 300.025,Z 399.836,A -85,B 0,C 180,E1 -18024.616,E2 -18024.616} C_VEL
LIN {X 0,Y 296.491,Z 392.827,A -85,B 0,C 180,E1 -18026.334,E2 -18026.334} C_VEL
LIN {X 0,Y 292.646,Z 386.058,A -85,B 0,C 180,E1 -18028.467,E2 -18028.467} C_VEL
LIN {X 0,Y 290.373,Z 382.334,A -85,B 0,C 180,E1 -18029.969,E2 -18029.969} C_VEL
LIN {X 0,Y 287.881,Z 378.803,A -85,B 0,C 180,E1 -18031.888,E2 -18031.888} C_VEL
LIN {X 0,Y 287.176,Z 377.47,A -85,B 0,C 180,E1 -18032.576,E2 -18032.576} C_VEL
LIN {X 0,Y 285.033,Z 374.954,A -85,B 0,C 180,E1 -18034.97,E2 -18034.97} C_VEL
LIN {X 0,Y 284.488,Z 373.954,A -85,B 0,C 180,E1 -18035.889,E2 -18035.889} C_VEL
LIN {X 0,Y 283.731,Z 373.099,A -85,B 0,C 180,E1 -18037.566,E2 -18037.566} C_VEL
LIN {X 0,Y 283.214,Z 373.341,A -85,B 0,C 180,E1 -18040.367,E2 -18040.367} C_VEL
LIN {X 0,Y 284.269,Z 375.751,A -85,B 0,C 180,E1 -18044.071,E2 -18044.071} C_VEL
LIN {X 0,Y 285.358,Z 377.12,A -85,B 0,C 180,E1 -18045.581,E2 -18045.581} C_VEL
LIN {X 0,Y 288.494,Z 382.35,A -85,B 0,C 180,E1 -18048.709,E2 -18048.709} C_VEL
LIN {X 0,Y 291.399,Z 387.11,A -85,B 0,C 180,E1 -18050.801,E2 -18050.801} C_VEL
LIN {X 0,Y 293.982,Z 398.739,A -85,B 0,C 180,E1 -18053.04,E2 -18053.04} C_VEL
LIN {X 0,Y 294.324,Z 402.183,A -85,B 0,C 180,E1 -18053.482,E2 -18053.482} C_VEL
LIN {X 0,Y 294.668,Z 420.144,A -85,B 0,C 180,E1 -18055.118,E2 -18055.118} C_VEL
LIN {X 0,Y 294.728,Z 442.083,A -85,B 0,C 180,E1 -18056.808,E2 -18056.808} C_VEL
LIN {X 0,Y 294.226,Z 459.992,A -85,B 0,C 180,E1 -18057.937,E2 -18057.937} C_VEL
LIN {X 0,Y 290.7,Z 490.658,A -85,B 0,C 180,E1 -18059.202,E2 -18059.202} C_VEL
LIN {X 0,Y 288.16,Z 505.012,A -85,B 0,C 180,E1 -18060.001,E2 -18060.001} C_VEL
LIN {X 0,Y 285.045,Z 518.996,A -85,B 0,C 180,E1 -18061.061,E2 -18061.061} C_VEL
LIN {X 0,Y 281.647,Z 531.549,A -85,B 0,C 180,E1 -18062.305,E2 -18062.305} C_VEL
LIN {X 0,Y 278.138,Z 542.992,A -85,B 0,C 180,E1 -18063.756,E2 -18063.756} C_VEL
LIN {X 0,Y 274.706,Z 553.582,A -85,B 0,C 180,E1 -18065.434,E2 -18065.434} C_VEL
LIN {X 0,Y 271.812,Z 562.37,A -85,B 0,C 180,E1 -18067.179,E2 -18067.179} C_VEL
LIN {X 0,Y 268.637,Z 571.201,A -85,B 0,C 180,E1 -18069.318,E2 -18069.318} C_VEL
LIN {X 0,Y 266.141,Z 578.543,A -85,B 0,C 180,E1 -18071.525,E2 -18071.525} C_VEL
LIN {X 0,Y 264.363,Z 584.549,A -85,B 0,C 180,E1 -18073.791,E2 -18073.791} C_VEL
LIN {X 0,Y 262.942,Z 589.414,A -85,B 0,C 180,E1 -18076.08,E2 -18076.08} C_VEL
LIN {X 0,Y 262.05,Z 593.224,A -85,B 0,C 180,E1 -18078.396,E2 -18078.396} C_VEL
LIN {X 0,Y 261.707,Z 596.055,A -85,B 0,C 180,E1 -18080.727,E2 -18080.727} C_VEL
LIN {X 0,Y 261.87,Z 598.061,A -85,B 0,C 180,E1 -18083.22,E2 -18083.22} C_VEL
LIN {X 0,Y 262.212,Z 598.907,A -85,B 0,C 180,E1 -18085.388,E2 -18085.388} C_VEL
LIN {X 0,Y 262.477,Z 598.991,A -85,B 0,C 180,E1 -18086.93,E2 -18086.93} C_VEL
LIN {X 0,Y 263.145,Z 598.101,A -85,B 0,C 180,E1 -18089.808,E2 -18089.808} C_VEL
LIN {X 0,Y 262.788,Z 599.23,A -85,B 0,C 180,E1 -18091.532,E2 -18091.532} C_VEL
LIN {X 0,Y 262.453,Z 599.757,A -85,B 0,C 180,E1 -18093.07,E2 -18093.07} C_VEL
LIN {X 0,Y 262.148,Z 599.851,A -85,B 0,C 180,E1 -18094.613,E2 -18094.613} C_VEL
LIN {X 0,Y 261.811,Z 599.257,A -85,B 0,C 180,E1 -18096.669,E2 -18096.669} C_VEL
LIN {X 0,Y 261.655,Z 597.477,A -85,B 0,C 180,E1 -18099.274,E2 -18099.274} C_VEL
LIN {X 0,Y 262.226,Z 593.89,A -85,B 0,C 180,E1 -18102.381,E2 -18102.381} C_VEL
LIN {X 0,Y 263.309,Z 590.076,A -85,B 0,C 180,E1 -18104.688,E2 -18104.688} C_VEL
LIN {X 0,Y 264.935,Z 585.257,A -85,B 0,C 180,E1 -18106.966,E2 -18106.966} C_VEL
LIN {X 0,Y 267.424,Z 578.258,A -85,B 0,C 180,E1 -18109.577,E2 -18109.577} C_VEL
LIN {X 0,Y 270.801,Z 569.516,A -85,B 0,C 180,E1 -18112.105,E2 -18112.105} C_VEL
LIN {X 0,Y 274.303,Z 560.416,A -85,B 0,C 180,E1 -18114.201,E2 -18114.201} C_VEL
LIN {X 0,Y 278.005,Z 550.38,A -85,B 0,C 180,E1 -18116.055,E2 -18116.055} C_VEL
LIN {X 0,Y 281.861,Z 539.497,A -85,B 0,C 180,E1 -18117.671,E2 -18117.671} C_VEL
LIN {X 0,Y 286.205,Z 526.222,A -85,B 0,C 180,E1 -18119.212,E2 -18119.212} C_VEL
LIN {X 0,Y 289.837,Z 513.171,A -85,B 0,C 180,E1 -18120.41,E2 -18120.41} C_VEL
LIN {X 0,Y 293.377,Z 498.545,A -85,B 0,C 180,E1 -18121.402,E2 -18121.402} C_VEL
LIN {X 0,Y 296.104,Z 483.49,A -85,B 0,C 180,E1 -18122.178,E2 -18122.178} C_VEL
LIN {X 0,Y 299.415,Z 457.925,A -85,B 0,C 180,E1 -18123.308,E2 -18123.308} C_VEL
LIN {X 0,Y 300.133,Z 445.058,A -85,B 0,C 180,E1 -18124.194,E2 -18124.194} C_VEL
LIN {X 0,Y 300.268,Z 429.673,A -85,B 0,C 180,E1 -18125.601,E2 -18125.601} C_VEL
LIN {X 0,Y 300.02,Z 416.667,A -85,B 0,C 180,E1 -18127.076,E2 -18127.076} C_VEL
LIN {X 0,Y 299.796,Z 414.295,A -85,B 0,C 180,E1 -18127.45,E2 -18127.45} C_VEL
LIN {X 0,Y 297.835,Z 407.7,A -85,B 0,C 180,E1 -18129.282,E2 -18129.282} C_VEL
LIN {X 0,Y 295.395,Z 399.638,A -85,B 0,C 180,E1 -18132.476,E2 -18132.476} C_VEL
LIN {X 0,Y 294.347,Z 395.801,A -85,B 0,C 180,E1 -18135.08,E2 -18135.08} C_VEL
LIN {X 0,Y 294.421,Z 393.308,A -85,B 0,C 180,E1 -18137.905,E2 -18137.905} C_VEL
LIN {X 0,Y 294.708,Z 392.908,A -85,B 0,C 180,E1 -18138.827,E2 -18138.827} C_VEL
LIN {X 0,Y 296.582,Z 393.362,A -85,B 0,C 180,E1 -18141.966,E2 -18141.966} C_VEL
LIN {X 0,Y 297.764,Z 393.99,A -85,B 0,C 180,E1 -18143.162,E2 -18143.162} C_VEL
LIN {X 0,Y 299.817,Z 395.941,A -85,B 0,C 180,E1 -18144.918,E2 -18144.918} C_VEL
LIN {X 0,Y 302.391,Z 399.134,A -85,B 0,C 180,E1 -18146.719,E2 -18146.719} C_VEL
LIN {X 0,Y 303.771,Z 401.111,A -85,B 0,C 180,E1 -18147.568,E2 -18147.568} C_VEL
LIN {X 0,Y 305.53,Z 404.877,A -85,B 0,C 180,E1 -18148.666,E2 -18148.666} C_VEL
LIN {X 0,Y 300.884,Z 436.259,A -85,B 0,C 180,E1 -18150.047,E2 -18150.047} C_VEL
LIN {X 0,Y 298.676,Z 454.201,A -85,B 0,C 180,E1 -18151.027,E2 -18151.027} C_VEL
LIN {X 0,Y 296.571,Z 467.315,A -85,B 0,C 180,E1 -18152.015,E2 -18152.015} C_VEL
LIN {X 0,Y 293.668,Z 480.804,A -85,B 0,C 180,E1 -18153.338,E2 -18153.338} C_VEL
LIN {X 0,Y 290.637,Z 492.143,A -85,B 0,C 180,E1 -18154.773,E2 -18154.773} C_VEL
LIN {X 0,Y 287.658,Z 501.547,A -85,B 0,C 180,E1 -18156.226,E2 -18156.226} C_VEL
LIN {X 0,Y 284.533,Z 510.209,A -85,B 0,C 180,E1 -18157.871,E2 -18157.871} C_VEL
LIN {X 0,Y 281.04,Z 518.713,A -85,B 0,C 180,E1 -18159.888,E2 -18159.888} C_VEL
LIN {X 0,Y 277.878,Z 525.595,A -85,B 0,C 180,E1 -18161.951,E2 -18161.951} C_VEL
LIN {X 0,Y 275.403,Z 530.275,A -85,B 0,C 180,E1 -18163.697,E2 -18163.697} C_VEL
LIN {X 0,Y 272.756,Z 534.79,A -85,B 0,C 180,E1 -18165.83,E2 -18165.83} C_VEL
LIN {X 0,Y 270.388,Z 538.204,A -85,B 0,C 180,E1 -18167.998,E2 -18167.998} C_VEL
LIN {X 0,Y 269.038,Z 539.896,A -85,B 0,C 180,E1 -18169.463,E2 -18169.463} C_VEL
LIN {X 0,Y 267.761,Z 541.152,A -85,B 0,C 180,E1 -18170.938,E2 -18170.938} C_VEL
LIN {X 0,Y 266.686,Z 541.994,A -85,B 0,C 180,E1 -18172.428,E2 -18172.428} C_VEL
LIN {X 0,Y 265.748,Z 542.426,A -85,B 0,C 180,E1 -18173.927,E2 -18173.927} C_VEL
LIN {X 0,Y 264.902,Z 542.41,A -85,B 0,C 180,E1 -18175.434,E2 -18175.434} C_VEL
LIN {X 0,Y 264.267,Z 541.98,A -85,B 0,C 180,E1 -18176.95,E2 -18176.95} C_VEL
LIN {X 0,Y 263.722,Z 541.153,A -85,B 0,C 180,E1 -18178.472,E2 -18178.472} C_VEL
LIN {X 0,Y 263.321,Z 539.888,A -85,B 0,C 180,E1 -18179.999,E2 -18179.999} C_VEL
LIN {X 0,Y 262.665,Z 537.191,A -85,B 0,C 180,E1 -18182.299,E2 -18182.299} C_VEL
LIN {X 0,Y 262.626,Z 533.442,A -85,B 0,C 180,E1 -18184.604,E2 -18184.604} C_VEL
LIN {X 0,Y 262.796,Z 527.609,A -85,B 0,C 180,E1 -18187.306,E2 -18187.306} C_VEL
LIN {X 0,Y 263.073,Z 521.282,A -85,B 0,C 180,E1 -18189.611,E2 -18189.611} C_VEL
LIN {X 0,Y 263.505,Z 513.397,A -85,B 0,C 180,E1 -18191.928,E2 -18191.928} C_VEL
LIN {X 0,Y 264.19,Z 503.626,A -85,B 0,C 180,E1 -18194.244,E2 -18194.244} C_VEL
LIN {X 0,Y 264.939,Z 493.614,A -85,B 0,C 180,E1 -18196.172,E2 -18196.172} C_VEL
LIN {X 0,Y 265.734,Z 482.552,A -85,B 0,C 180,E1 -18197.911,E2 -18197.911} C_VEL
LIN {X 0,Y 266.606,Z 470.553,A -85,B 0,C 180,E1 -18199.438,E2 -18199.438} C_VEL
LIN {X 0,Y 267.299,Z 456.985,A -85,B 0,C 180,E1 -18200.79,E2 -18200.79} C_VEL
LIN {X 0,Y 268.009,Z 443.468,A -85,B 0,C 180,E1 -18201.79,E2 -18201.79} C_VEL
LIN {X 0,Y 268.322,Z 429.45,A -85,B 0,C 180,E1 -18202.523,E2 -18202.523} C_VEL
LIN {X 0,Y 270.106,Z 375.25,A -85,B 0,C 180,E1 -18204.702,E2 -18204.702} C_VEL
LIN {X 0,Y 270.175,Z 372.04,A -85,B 0,C 180,E1 -18204.834,E2 -18204.834} C_VEL
LIN {X 0,Y 263.276,Z 348.688,A -85,B 0,C 180,E1 -18206.149,E2 -18206.149} C_VEL
LIN {X 0,Y 263.15,Z 348.703,A -85,B 0,C 180,E1 -18210.492,E2 -18210.492} C_VEL
LIN {X 0,Y 263.15,Z 348.704,A -85,B 0,C 180,E1 -18214.114,E2 -18214.114} C_VEL
LIN {X 0,Y 263.157,Z 348.701,A -85,B 0,C 180,E1 -18217.896,E2 -18217.896} C_VEL
LIN {X 0,Y 263.123,Z 348.707,A -85,B 0,C 180,E1 -18221.892,E2 -18221.892} C_VEL
LIN {X 0,Y 263.126,Z 348.706,A -85,B 0,C 180,E1 -18226.149,E2 -18226.149} C_VEL
LIN {X 0,Y 263.113,Z 348.709,A -85,B 0,C 180,E1 -18230.129,E2 -18230.129} C_VEL
LIN {X 0,Y 263.185,Z 348.699,A -85,B 0,C 180,E1 -18234.022,E2 -18234.022} C_VEL
LIN {X 0,Y 263.131,Z 348.705,A -85,B 0,C 180,E1 -18237.712,E2 -18237.712} C_VEL
LIN {X 0,Y 263.193,Z 348.698,A -85,B 0,C 180,E1 -18241.785,E2 -18241.785} C_VEL
LIN {X 0,Y 263.223,Z 348.694,A -85,B 0,C 180,E1 -18245.2,E2 -18245.2} C_VEL
LIN {X 0,Y 263.261,Z 348.69,A -85,B 0,C 180,E1 -18249.693,E2 -18249.693} C_VEL
LIN {X 0,Y 263.348,Z 348.682,A -85,B 0,C 180,E1 -18254.522,E2 -18254.522} C_VEL
LIN {X 0,Y 263.371,Z 348.675,A -85,B 0,C 180,E1 -18259.234,E2 -18259.234} C_VEL
LIN {X 0,Y 263.57,Z 348.653,A -85,B 0,C 180,E1 -18262.339,E2 -18262.339} C_VEL
LIN {X 0,Y 263.749,Z 348.631,A -85,B 0,C 180,E1 -18268.473,E2 -18268.473} C_VEL
LIN {X 0,Y 263.749,Z 348.628,A -85,B 0,C 180,E1 -18271.527,E2 -18271.527} C_VEL
LIN {X 0,Y 263.571,Z 348.65,A -85,B 0,C 180,E1 -18277.662,E2 -18277.662} C_VEL
LIN {X 0,Y 263.372,Z 348.677,A -85,B 0,C 180,E1 -18280.766,E2 -18280.766} C_VEL
LIN {X 0,Y 263.349,Z 348.678,A -85,B 0,C 180,E1 -18285.478,E2 -18285.478} C_VEL
LIN {X 0,Y 263.262,Z 348.694,A -85,B 0,C 180,E1 -18290.307,E2 -18290.307} C_VEL
LIN {X 0,Y 263.207,Z 348.694,A -85,B 0,C 180,E1 -18295.292,E2 -18295.292} C_VEL
LIN {X 0,Y 263.164,Z 348.703,A -85,B 0,C 180,E1 -18298.732,E2 -18298.732} C_VEL
LIN {X 0,Y 263.132,Z 348.708,A -85,B 0,C 180,E1 -18302.289,E2 -18302.289} C_VEL
LIN {X 0,Y 263.187,Z 348.701,A -85,B 0,C 180,E1 -18305.979,E2 -18305.979} C_VEL
LIN {X 0,Y 263.114,Z 348.711,A -85,B 0,C 180,E1 -18309.872,E2 -18309.872} C_VEL
LIN {X 0,Y 263.122,Z 348.709,A -85,B 0,C 180,E1 -18313.985,E2 -18313.985} C_VEL
LIN {X 0,Y 263.124,Z 348.708,A -85,B 0,C 180,E1 -18318.407,E2 -18318.407} C_VEL
LIN {X 0,Y 263.194,Z 348.697,A -85,B 0,C 180,E1 -18323.234,E2 -18323.234} C_VEL
LIN {X 0,Y 263.185,Z 348.7,A -85,B 0,C 180,E1 -18327.44,E2 -18327.44} C_VEL
LIN {X 0,Y 270.768,Z 372.442,A -85,B 0,C 180,E1 -18328.78,E2 -18328.78} C_VEL
LIN {X 0,Y 268.879,Z 433.688,A -85,B 0,C 180,E1 -18331.136,E2 -18331.136} C_VEL
LIN {X 0,Y 268.448,Z 446.863,A -85,B 0,C 180,E1 -18331.886,E2 -18331.886} C_VEL
LIN {X 0,Y 267.741,Z 460.819,A -85,B 0,C 180,E1 -18333.009,E2 -18333.009} C_VEL
LIN {X 0,Y 266.966,Z 472.715,A -85,B 0,C 180,E1 -18334.256,E2 -18334.256} C_VEL
LIN {X 0,Y 266.086,Z 484.569,A -85,B 0,C 180,E1 -18335.834,E2 -18335.834} C_VEL
LIN {X 0,Y 265.163,Z 495.491,A -85,B 0,C 180,E1 -18337.626,E2 -18337.626} C_VEL
LIN {X 0,Y 264.296,Z 506.013,A -85,B 0,C 180,E1 -18339.777,E2 -18339.777} C_VEL
LIN {X 0,Y 263.662,Z 513.937,A -85,B 0,C 180,E1 -18341.749,E2 -18341.749} C_VEL
LIN {X 0,Y 263.165,Z 521.417,A -85,B 0,C 180,E1 -18344.032,E2 -18344.032} C_VEL
LIN {X 0,Y 262.841,Z 526.876,A -85,B 0,C 180,E1 -18346.076,E2 -18346.076} C_VEL
LIN {X 0,Y 262.682,Z 531.892,A -85,B 0,C 180,E1 -18348.425,E2 -18348.425} C_VEL
LIN {X 0,Y 262.778,Z 535.727,A -85,B 0,C 180,E1 -18350.767,E2 -18350.767} C_VEL
LIN {X 0,Y 262.977,Z 537.71,A -85,B 0,C 180,E1 -18352.322,E2 -18352.322} C_VEL
LIN {X 0,Y 263.194,Z 539.198,A -85,B 0,C 180,E1 -18353.869,E2 -18353.869} C_VEL
LIN {X 0,Y 263.499,Z 540.264,A -85,B 0,C 180,E1 -18355.411,E2 -18355.411} C_VEL
LIN {X 0,Y 264.131,Z 540.941,A -85,B 0,C 180,E1 -18357.2,E2 -18357.2} C_VEL
LIN {X 0,Y 265.459,Z 540.854,A -85,B 0,C 180,E1 -18360.001,E2 -18360.001} C_VEL
LIN {X 0,Y 266.333,Z 540.22,A -85,B 0,C 180,E1 -18361.513,E2 -18361.513} C_VEL
LIN {X 0,Y 267.882,Z 538.411,A -85,B 0,C 180,E1 -18363.727,E2 -18363.727} C_VEL
LIN {X 0,Y 268.208,Z 537.245,A -85,B 0,C 180,E1 -18364.964,E2 -18364.964} C_VEL
LIN {X 0,Y 267.293,Z 535.206,A -85,B 0,C 180,E1 -18367.035,E2 -18367.035} C_VEL
LIN {X 0,Y 266.646,Z 532.527,A -85,B 0,C 180,E1 -18369.072,E2 -18369.072} C_VEL
LIN {X 0,Y 267.361,Z 530.257,A -85,B 0,C 180,E1 -18370.227,E2 -18370.227} C_VEL
LIN {X 0,Y 270.225,Z 524.617,A -85,B 0,C 180,E1 -18372.391,E2 -18372.391} C_VEL
LIN {X 0,Y 273.396,Z 517.537,A -85,B 0,C 180,E1 -18374.516,E2 -18374.516} C_VEL
LIN {X 0,Y 276.236,Z 510.323,A -85,B 0,C 180,E1 -18376.253,E2 -18376.253} C_VEL
LIN {X 0,Y 279.888,Z 499.744,A -85,B 0,C 180,E1 -18378.294,E2 -18378.294} C_VEL
LIN {X 0,Y 282.784,Z 490.005,A -85,B 0,C 180,E1 -18379.794,E2 -18379.794} C_VEL
LIN {X 0,Y 285.446,Z 479.306,A -85,B 0,C 180,E1 -18381.106,E2 -18381.106} C_VEL
LIN {X 0,Y 288.081,Z 465.978,A -85,B 0,C 180,E1 -18382.408,E2 -18382.408} C_VEL
LIN {X 0,Y 290.104,Z 452.169,A -85,B 0,C 180,E1 -18383.42,E2 -18383.42} C_VEL
LIN {X 0,Y 291.884,Z 434.875,A -85,B 0,C 180,E1 -18384.298,E2 -18384.298} C_VEL
LIN {X 0,Y 295.794,Z 403.36,A -85,B 0,C 180,E1 -18385.657,E2 -18385.657} C_VEL
LIN {X 0,Y 292.613,Z 396.998,A -85,B 0,C 180,E1 -18387.37,E2 -18387.37} C_VEL
LIN {X 0,Y 289.588,Z 391.592,A -85,B 0,C 180,E1 -18389.244,E2 -18389.244} C_VEL
LIN {X 0,Y 287.583,Z 388.189,A -85,B 0,C 180,E1 -18390.689,E2 -18390.689} C_VEL
LIN {X 0,Y 285.546,Z 384.896,A -85,B 0,C 180,E1 -18392.461,E2 -18392.461} C_VEL
LIN {X 0,Y 285.02,Z 384.007,A -85,B 0,C 180,E1 -18393.031,E2 -18393.031} C_VEL
LIN {X 0,Y 283.082,Z 381.341,A -85,B 0,C 180,E1 -18395.498,E2 -18395.498} C_VEL
LIN {X 0,Y 282.178,Z 380.094,A -85,B 0,C 180,E1 -18397.404,E2 -18397.404} C_VEL
LIN {X 0,Y 281.597,Z 380.16,A -85,B 0,C 180,E1 -18400.152,E2 -18400.152} C_VEL
LIN {X 0,Y 282.547,Z 382.605,A -85,B 0,C 180,E1 -18403.937,E2 -18403.937} C_VEL
LIN {X 0,Y 283.475,Z 383.781,A -85,B 0,C 180,E1 -18405.259,E2 -18405.259} C_VEL
LIN {X 0,Y 286.232,Z 388.723,A -85,B 0,C 180,E1 -18408.275,E2 -18408.275} C_VEL
LIN {X 0,Y 288.622,Z 392.918,A -85,B 0,C 180,E1 -18410.156,E2 -18410.156} C_VEL
LIN {X 0,Y 290.619,Z 403.143,A -85,B 0,C 180,E1 -18412.168,E2 -18412.168} C_VEL
LIN {X 0,Y 290.789,Z 407.967,A -85,B 0,C 180,E1 -18412.712,E2 -18412.712} C_VEL
LIN {X 0,Y 290.778,Z 426.407,A -85,B 0,C 180,E1 -18414.385,E2 -18414.385} C_VEL
LIN {X 0,Y 290.43,Z 446.67,A -85,B 0,C 180,E1 -18415.944,E2 -18415.944} C_VEL
LIN {X 0,Y 289.747,Z 461.73,A -85,B 0,C 180,E1 -18416.885,E2 -18416.885} C_VEL
LIN {X 0,Y 286.107,Z 490.618,A -85,B 0,C 180,E1 -18418.12,E2 -18418.12} C_VEL
LIN {X 0,Y 283.392,Z 504.78,A -85,B 0,C 180,E1 -18418.926,E2 -18418.926} C_VEL
LIN {X 0,Y 279.924,Z 519.214,A -85,B 0,C 180,E1 -18420.066,E2 -18420.066} C_VEL
LIN {X 0,Y 275.921,Z 532.723,A -85,B 0,C 180,E1 -18421.472,E2 -18421.472} C_VEL
LIN {X 0,Y 271.896,Z 544.855,A -85,B 0,C 180,E1 -18423.106,E2 -18423.106} C_VEL
LIN {X 0,Y 268.342,Z 554.825,A -85,B 0,C 180,E1 -18424.811,E2 -18424.811} C_VEL
LIN {X 0,Y 264.761,Z 564.746,A -85,B 0,C 180,E1 -18426.95,E2 -18426.95} C_VEL
LIN {X 0,Y 261.552,Z 572.945,A -85,B 0,C 180,E1 -18429.143,E2 -18429.143} C_VEL
LIN {X 0,Y 258.998,Z 579.815,A -85,B 0,C 180,E1 -18431.448,E2 -18431.448} C_VEL
LIN {X 0,Y 256.92,Z 586.128,A -85,B 0,C 180,E1 -18434.124,E2 -18434.124} C_VEL
LIN {X 0,Y 255.65,Z 590.409,A -85,B 0,C 180,E1 -18436.486,E2 -18436.486} C_VEL
LIN {X 0,Y 254.868,Z 593.703,A -85,B 0,C 180,E1 -18438.87,E2 -18438.87} C_VEL
LIN {X 0,Y 254.66,Z 595.386,A -85,B 0,C 180,E1 -18440.468,E2 -18440.468} C_VEL
LIN {X 0,Y 254.871,Z 597.49,A -85,B 0,C 180,E1 -18443.667,E2 -18443.667} C_VEL
LIN {X 0,Y 255.147,Z 597.93,A -85,B 0,C 180,E1 -18445.26,E2 -18445.26} C_VEL
LIN {X 0,Y 255.43,Z 597.917,A -85,B 0,C 180,E1 -18446.845,E2 -18446.845} C_VEL
LIN {X 0,Y 256.21,Z 596.751,A -85,B 0,C 180,E1 -18449.902,E2 -18449.902} C_VEL
LIN {X 0,Y 255.789,Z 597.946,A -85,B 0,C 180,E1 -18451.574,E2 -18451.574} C_VEL
LIN {X 0,Y 255.426,Z 598.555,A -85,B 0,C 180,E1 -18453.154,E2 -18453.154} C_VEL
LIN {X 0,Y 255.104,Z 598.732,A -85,B 0,C 180,E1 -18454.741,E2 -18454.741} C_VEL
LIN {X 0,Y 254.766,Z 598.373,A -85,B 0,C 180,E1 -18456.729,E2 -18456.729} C_VEL
LIN {X 0,Y 254.614,Z 596.739,A -85,B 0,C 180,E1 -18459.533,E2 -18459.533} C_VEL
LIN {X 0,Y 255.255,Z 593.365,A -85,B 0,C 180,E1 -18462.724,E2 -18462.724} C_VEL
LIN {X 0,Y 256.395,Z 589.785,A -85,B 0,C 180,E1 -18465.094,E2 -18465.094} C_VEL
LIN {X 0,Y 258.36,Z 584.388,A -85,B 0,C 180,E1 -18467.806,E2 -18467.806} C_VEL
LIN {X 0,Y 261.207,Z 577.497,A -85,B 0,C 180,E1 -18470.474,E2 -18470.474} C_VEL
LIN {X 0,Y 264.864,Z 568.911,A -85,B 0,C 180,E1 -18473.04,E2 -18473.04} C_VEL
LIN {X 0,Y 268.588,Z 559.989,A -85,B 0,C 180,E1 -18475.164,E2 -18475.164} C_VEL
LIN {X 0,Y 272.906,Z 549.238,A -85,B 0,C 180,E1 -18477.2,E2 -18477.2} C_VEL
LIN {X 0,Y 277.014,Z 538.44,A -85,B 0,C 180,E1 -18478.819,E2 -18478.819} C_VEL
LIN {X 0,Y 281.582,Z 525.385,A -85,B 0,C 180,E1 -18480.359,E2 -18480.359} C_VEL
LIN {X 0,Y 285.964,Z 510.764,A -85,B 0,C 180,E1 -18481.69,E2 -18481.69} C_VEL
LIN {X 0,Y 289.729,Z 495.938,A -85,B 0,C 180,E1 -18482.665,E2 -18482.665} C_VEL
LIN {X 0,Y 292.376,Z 481.725,A -85,B 0,C 180,E1 -18483.409,E2 -18483.409} C_VEL
LIN {X 0,Y 295.553,Z 458.872,A -85,B 0,C 180,E1 -18484.445,E2 -18484.445} C_VEL
LIN {X 0,Y 296.429,Z 446.151,A -85,B 0,C 180,E1 -18485.365,E2 -18485.365} C_VEL
LIN {X 0,Y 296.799,Z 431.432,A -85,B 0,C 180,E1 -18486.771,E2 -18486.771} C_VEL
LIN {X 0,Y 296.837,Z 419.533,A -85,B 0,C 180,E1 -18488.184,E2 -18488.184} C_VEL
LIN {X 0,Y 295.209,Z 413.338,A -85,B 0,C 180,E1 -18489.966,E2 -18489.966} C_VEL
LIN {X 0,Y 293.278,Z 405.926,A -85,B 0,C 180,E1 -18492.981,E2 -18492.981} C_VEL
LIN {X 0,Y 292.5,Z 402.245,A -85,B 0,C 180,E1 -18495.598,E2 -18495.598} C_VEL
LIN {X 0,Y 292.726,Z 400.122,A -85,B 0,C 180,E1 -18498.097,E2 -18498.097} C_VEL
LIN {X 0,Y 293.303,Z 399.798,A -85,B 0,C 180,E1 -18499.686,E2 -18499.686} C_VEL
LIN {X 0,Y 295.699,Z 400.588,A -85,B 0,C 180,E1 -18502.865,E2 -18502.865} C_VEL
LIN {X 0,Y 297.734,Z 402.701,A -85,B 0,C 180,E1 -18504.724,E2 -18504.724} C_VEL
LIN {X 0,Y 300.683,Z 406.43,A -85,B 0,C 180,E1 -18506.825,E2 -18506.825} C_VEL
LIN {X 0,Y 301.808,Z 408.891,A -85,B 0,C 180,E1 -18507.616,E2 -18507.616} C_VEL
LIN {X 0,Y 297.196,Z 438.117,A -85,B 0,C 180,E1 -18508.935,E2 -18508.935} C_VEL
LIN {X 0,Y 294.855,Z 455.507,A -85,B 0,C 180,E1 -18509.902,E2 -18509.902} C_VEL
LIN {X 0,Y 292.526,Z 468.759,A -85,B 0,C 180,E1 -18510.916,E2 -18510.916} C_VEL
LIN {X 0,Y 289.636,Z 481.251,A -85,B 0,C 180,E1 -18512.153,E2 -18512.153} C_VEL
